LIN {X 0,Y 411.201,Z 389.266,A -85,B 0,C 180,E1 -10586.873,E2 -10586.873} C_VEL
LIN {X 0,Y 411.226,Z 389.263,A -85,B 0,C 180,E1 -10590.644,E2 -10590.644} C_VEL
LIN {X 0,Y 411.231,Z 389.26,A -85,B 0,C 180,E1 -10593.619,E2 -10593.619} C_VEL
LIN {X 0,Y 411.195,Z 389.267,A -85,B 0,C 180,E1 -10596.852,E2 -10596.852} C_VEL
LIN {X 0,Y 411.206,Z 389.262,A -85,B 0,C 180,E1 -10600.05,E2 -10600.05} C_VEL
LIN {X 0,Y 411.255,Z 389.259,A -85,B 0,C 180,E1 -10603.131,E2 -10603.131} C_VEL
LIN {X 0,Y 411.296,Z 389.255,A -85,B 0,C 180,E1 -10606.896,E2 -10606.896} C_VEL
LIN {X 0,Y 411.285,Z 389.254,A -85,B 0,C 180,E1 -10610.161,E2 -10610.161} C_VEL
LIN {X 0,Y 411.447,Z 389.234,A -85,B 0,C 180,E1 -10613.133,E2 -10613.133} C_VEL
LIN {X 0,Y 411.303,Z 389.252,A -85,B 0,C 180,E1 -10615.099,E2 -10615.099} C_VEL
LIN {X 0,Y 411.505,Z 389.226,A -85,B 0,C 180,E1 -10618.043,E2 -10618.043} C_VEL
LIN {X 0,Y 411.635,Z 389.21,A -85,B 0,C 180,E1 -10620,E2 -10620} C_VEL
LIN {X 0,Y 411.458,Z 389.233,A -85,B 0,C 180,E1 -10622.937,E2 -10622.937} C_VEL
LIN {X 0,Y 411.452,Z 389.235,A -85,B 0,C 180,E1 -10626.867,E2 -10626.867} C_VEL
LIN {X 0,Y 411.286,Z 389.253,A -85,B 0,C 180,E1 -10629.839,E2 -10629.839} C_VEL
LIN {X 0,Y 411.297,Z 389.252,A -85,B 0,C 180,E1 -10633.104,E2 -10633.104} C_VEL
LIN {X 0,Y 411.249,Z 389.259,A -85,B 0,C 180,E1 -10636.889,E2 -10636.889} C_VEL
LIN {X 0,Y 411.223,Z 389.262,A -85,B 0,C 180,E1 -10639.987,E2 -10639.987} C_VEL
LIN {X 0,Y 411.196,Z 389.264,A -85,B 0,C 180,E1 -10643.148,E2 -10643.148} C_VEL
LIN {X 0,Y 411.231,Z 389.263,A -85,B 0,C 180,E1 -10646.382,E2 -10646.382} C_VEL
LIN {X 0,Y 411.194,Z 389.265,A -85,B 0,C 180,E1 -10649.713,E2 -10649.713} C_VEL
LIN {X 0,Y 411.201,Z 389.263,A -85,B 0,C 180,E1 -10653.157,E2 -10653.157} C_VEL
LIN {X 0,Y 411.191,Z 389.268,A -85,B 0,C 180,E1 -10656.554,E2 -10656.554} C_VEL
LIN {X 0,Y 411.224,Z 389.262,A -85,B 0,C 180,E1 -10659.731,E2 -10659.731} C_VEL
LIN {X 0,Y 411.173,Z 389.266,A -85,B 0,C 180,E1 -10663.134,E2 -10663.134} C_VEL
LIN {X 0,Y 411.165,Z 389.27,A -85,B 0,C 180,E1 -10665.882,E2 -10665.882} C_VEL
LIN {X 0,Y 411.162,Z 389.269,A -85,B 0,C 180,E1 -10668.772,E2 -10668.772} C_VEL
LIN {X 0,Y 411.209,Z 389.265,A -85,B 0,C 180,E1 -10671.831,E2 -10671.831} C_VEL
LIN {X 0,Y 411.21,Z 389.261,A -85,B 0,C 180,E1 -10675.122,E2 -10675.122} C_VEL
LIN {X 0,Y 411.165,Z 389.272,A -85,B 0,C 180,E1 -10678.004,E2 -10678.004} C_VEL
LIN {X 0,Y 411.218,Z 389.262,A -85,B 0,C 180,E1 -10681.411,E2 -10681.411} C_VEL
LIN {X 0,Y 411.239,Z 389.26,A -85,B 0,C 180,E1 -10683.62,E2 -10683.62} C_VEL
LIN {X 0,Y 411.205,Z 389.262,A -85,B 0,C 180,E1 -10686.853,E2 -10686.853} C_VEL
LIN {X 0,Y 411.217,Z 389.265,A -85,B 0,C 180,E1 -10690.051,E2 -10690.051} C_VEL
LIN {X 0,Y 411.265,Z 389.255,A -85,B 0,C 180,E1 -10693.132,E2 -10693.132} C_VEL
LIN {X 0,Y 411.308,Z 389.249,A -85,B 0,C 180,E1 -10696.896,E2 -10696.896} C_VEL
LIN {X 0,Y 411.295,Z 389.253,A -85,B 0,C 180,E1 -10700.162,E2 -10700.162} C_VEL
LIN {X 0,Y 411.465,Z 389.23,A -85,B 0,C 180,E1 -10703.133,E2 -10703.133} C_VEL
LIN {X 0,Y 411.311,Z 389.25,A -85,B 0,C 180,E1 -10705.099,E2 -10705.099} C_VEL
LIN {X 0,Y 411.438,Z 389.238,A -85,B 0,C 180,E1 -10708.043,E2 -10708.043} C_VEL
LIN {X 0,Y 411.179,Z 389.27,A -85,B 0,C 180,E1 -10710,E2 -10710} C_VEL
LIN {X 0,Y 410.704,Z 389.33,A -85,B 0,C 180,E1 -10710.981,E2 -10710.981} C_VEL
LIN {X 0,Y 410.736,Z 392.015,A -85,B 0,C 180,E1 -10713.925,E2 -10713.925} C_VEL
LIN {X 0,Y 410.647,Z 395.045,A -85,B 0,C 180,E1 -10716.953,E2 -10716.953} C_VEL
LIN {X 0,Y 410.457,Z 397.926,A -85,B 0,C 180,E1 -10719.859,E2 -10719.859} C_VEL
LIN {X 0,Y 410.386,Z 401.01,A -85,B 0,C 180,E1 -10722.864,E2 -10722.864} C_VEL
LIN {X 0,Y 410.342,Z 402.843,A -85,B 0,C 180,E1 -10724.601,E2 -10724.601} C_VEL
LIN {X 0,Y 413.667,Z 416.138,A -85,B 0,C 180,E1 -10725.205,E2 -10725.205} C_VEL
LIN {X 0,Y 415.457,Z 424.901,A -85,B 0,C 180,E1 -10725.704,E2 -10725.704} C_VEL
LIN {X 0,Y 415.437,Z 425.566,A -85,B 0,C 180,E1 -10725.74,E2 -10725.74} C_VEL
LIN {X 0,Y 414.599,Z 431.128,A -85,B 0,C 180,E1 -10726.033,E2 -10726.033} C_VEL
LIN {X 0,Y 411.37,Z 439.883,A -85,B 0,C 180,E1 -10726.51,E2 -10726.51} C_VEL
LIN {X 0,Y 408.025,Z 448.217,A -85,B 0,C 180,E1 -10727.08,E2 -10727.08} C_VEL
LIN {X 0,Y 406.998,Z 453.065,A -85,B 0,C 180,E1 -10727.509,E2 -10727.509} C_VEL
LIN {X 0,Y 406.214,Z 463.524,A -85,B 0,C 180,E1 -10728.667,E2 -10728.667} C_VEL
LIN {X 0,Y 405.456,Z 473.281,A -85,B 0,C 180,E1 -10730.019,E2 -10730.019} C_VEL
LIN {X 0,Y 404.761,Z 481.303,A -85,B 0,C 180,E1 -10731.385,E2 -10731.385} C_VEL
LIN {X 0,Y 404.171,Z 488.245,A -85,B 0,C 180,E1 -10732.838,E2 -10732.838} C_VEL
LIN {X 0,Y 403.811,Z 493.278,A -85,B 0,C 180,E1 -10734.142,E2 -10734.142} C_VEL
LIN {X 0,Y 403.461,Z 498.427,A -85,B 0,C 180,E1 -10735.816,E2 -10735.816} C_VEL
LIN {X 0,Y 403.282,Z 501.804,A -85,B 0,C 180,E1 -10737.279,E2 -10737.279} C_VEL
LIN {X 0,Y 403.135,Z 503.254,A -85,B 0,C 180,E1 -10738.079,E2 -10738.079} C_VEL
LIN {X 0,Y 402.957,Z 504.918,A -85,B 0,C 180,E1 -10739.301,E2 -10739.301} C_VEL
LIN {X 0,Y 402.872,Z 506.388,A -85,B 0,C 180,E1 -10741.263,E2 -10741.263} C_VEL
LIN {X 0,Y 402.872,Z 506.326,A -85,B 0,C 180,E1 -10743.138,E2 -10743.138} C_VEL
LIN {X 0,Y 403.019,Z 504.763,A -85,B 0,C 180,E1 -10745.132,E2 -10745.132} C_VEL
LIN {X 0,Y 403.253,Z 502.375,A -85,B 0,C 180,E1 -10746.707,E2 -10746.707} C_VEL
LIN {X 0,Y 403.549,Z 498.622,A -85,B 0,C 180,E1 -10748.399,E2 -10748.399} C_VEL
LIN {X 0,Y 403.946,Z 493.53,A -85,B 0,C 180,E1 -10750.071,E2 -10750.071} C_VEL
LIN {X 0,Y 404.465,Z 487.306,A -85,B 0,C 180,E1 -10751.654,E2 -10751.654} C_VEL
LIN {X 0,Y 405.136,Z 479.493,A -85,B 0,C 180,E1 -10753.232,E2 -10753.232} C_VEL
LIN {X 0,Y 405.807,Z 471.524,A -85,B 0,C 180,E1 -10754.526,E2 -10754.526} C_VEL
LIN {X 0,Y 406.609,Z 461.592,A -85,B 0,C 180,E1 -10755.831,E2 -10755.831} C_VEL
LIN {X 0,Y 407.402,Z 450.84,A -85,B 0,C 180,E1 -10756.97,E2 -10756.97} C_VEL
LIN {X 0,Y 408.167,Z 439.572,A -85,B 0,C 180,E1 -10757.91,E2 -10757.91} C_VEL
LIN {X 0,Y 408.846,Z 427.215,A -85,B 0,C 180,E1 -10758.702,E2 -10758.702} C_VEL
LIN {X 0,Y 408.184,Z 422.977,A -85,B 0,C 180,E1 -10758.964,E2 -10758.964} C_VEL
LIN {X 0,Y 404.917,Z 410.066,A -85,B 0,C 180,E1 -10759.678,E2 -10759.678} C_VEL
LIN {X 0,Y 403.332,Z 404.392,A -85,B 0,C 180,E1 -10759.963,E2 -10759.963} C_VEL
LIN {X 0,Y 403.388,Z 400.813,A -85,B 0,C 180,E1 -10763.675,E2 -10763.675} C_VEL
LIN {X 0,Y 403.574,Z 397.329,A -85,B 0,C 180,E1 -10767.327,E2 -10767.327} C_VEL
LIN {X 0,Y 403.731,Z 394.082,A -85,B 0,C 180,E1 -10770.829,E2 -10770.829} C_VEL
LIN {X 0,Y 403.781,Z 390.974,A -85,B 0,C 180,E1 -10774.206,E2 -10774.206} C_VEL
LIN {X 0,Y 403.855,Z 390.182,A -85,B 0,C 180,E1 -10775.313,E2 -10775.313} C_VEL
LIN {X 0,Y 404.117,Z 390.153,A -85,B 0,C 180,E1 -10777.505,E2 -10777.505} C_VEL
LIN {X 0,Y 404.161,Z 390.144,A -85,B 0,C 180,E1 -10780.707,E2 -10780.707} C_VEL
LIN {X 0,Y 404.216,Z 390.135,A -85,B 0,C 180,E1 -10783.848,E2 -10783.848} C_VEL
LIN {X 0,Y 404.278,Z 390.129,A -85,B 0,C 180,E1 -10786.939,E2 -10786.939} C_VEL
LIN {X 0,Y 404.254,Z 390.13,A -85,B 0,C 180,E1 -10789.988,E2 -10789.988} C_VEL
LIN {X 0,Y 404.398,Z 390.112,A -85,B 0,C 180,E1 -10793.012,E2 -10793.012} C_VEL
LIN {X 0,Y 404.278,Z 390.125,A -85,B 0,C 180,E1 -10795.013,E2 -10795.013} C_VEL
LIN {X 0,Y 404.477,Z 390.104,A -85,B 0,C 180,E1 -10798.008,E2 -10798.008} C_VEL
LIN {X 0,Y 404.605,Z 390.084,A -85,B 0,C 180,E1 -10800,E2 -10800} C_VEL
LIN {X 0,Y 404.417,Z 390.11,A -85,B 0,C 180,E1 -10802.988,E2 -10802.988} C_VEL
LIN {X 0,Y 404.397,Z 390.112,A -85,B 0,C 180,E1 -10806.987,E2 -10806.987} C_VEL
LIN {X 0,Y 404.253,Z 390.13,A -85,B 0,C 180,E1 -10810.012,E2 -10810.012} C_VEL
LIN {X 0,Y 404.261,Z 390.128,A -85,B 0,C 180,E1 -10813.211,E2 -10813.211} C_VEL
LIN {X 0,Y 404.211,Z 390.135,A -85,B 0,C 180,E1 -10817.007,E2 -10817.007} C_VEL
LIN {X 0,Y 404.159,Z 390.142,A -85,B 0,C 180,E1 -10820.352,E2 -10820.352} C_VEL
LIN {X 0,Y 404.165,Z 390.143,A -85,B 0,C 180,E1 -10823.575,E2 -10823.575} C_VEL
LIN {X 0,Y 404.179,Z 390.14,A -85,B 0,C 180,E1 -10825.767,E2 -10825.767} C_VEL
LIN {X 0,Y 404.191,Z 390.14,A -85,B 0,C 180,E1 -10828,E2 -10828} C_VEL
LIN {X 0,Y 404.135,Z 390.146,A -85,B 0,C 180,E1 -10831.558,E2 -10831.558} C_VEL
LIN {X 0,Y 404.18,Z 390.142,A -85,B 0,C 180,E1 -10835.017,E2 -10835.017} C_VEL
LIN {X 0,Y 404.161,Z 390.144,A -85,B 0,C 180,E1 -10838.756,E2 -10838.756} C_VEL
LIN {X 0,Y 404.147,Z 390.144,A -85,B 0,C 180,E1 -10841.604,E2 -10841.604} C_VEL
LIN {X 0,Y 404.143,Z 390.145,A -85,B 0,C 180,E1 -10844.523,E2 -10844.523} C_VEL
LIN {X 0,Y 404.158,Z 390.285,A -85,B 0,C 180,E1 -10845.838,E2 -10845.838} C_VEL
LIN {X 0,Y 405.078,Z 395.076,A -85,B 0,C 180,E1 -10848.755,E2 -10848.755} C_VEL
LIN {X 0,Y 406.148,Z 401.144,A -85,B 0,C 180,E1 -10852.101,E2 -10852.101} C_VEL
LIN {X 0,Y 406.513,Z 404.837,A -85,B 0,C 180,E1 -10853.999,E2 -10853.999} C_VEL
LIN {X 0,Y 405.924,Z 411.076,A -85,B 0,C 180,E1 -10856.95,E2 -10856.95} C_VEL
LIN {X 0,Y 405.292,Z 418.116,A -85,B 0,C 180,E1 -10860.115,E2 -10860.115} C_VEL
LIN {X 0,Y 404.69,Z 426.478,A -85,B 0,C 180,E1 -10863.715,E2 -10863.715} C_VEL
LIN {X 0,Y 404.135,Z 435.633,A -85,B 0,C 180,E1 -10867.506,E2 -10867.506} C_VEL
LIN {X 0,Y 403.824,Z 443.566,A -85,B 0,C 180,E1 -10870.691,E2 -10870.691} C_VEL
LIN {X 0,Y 403.621,Z 447.012,A -85,B 0,C 180,E1 -10872.063,E2 -10872.063} C_VEL
LIN {X 0,Y 405.834,Z 460.859,A -85,B 0,C 180,E1 -10872.593,E2 -10872.593} C_VEL
LIN {X 0,Y 407.534,Z 473.33,A -85,B 0,C 180,E1 -10873.255,E2 -10873.255} C_VEL
LIN {X 0,Y 407.967,Z 477.581,A -85,B 0,C 180,E1 -10873.516,E2 -10873.516} C_VEL
LIN {X 0,Y 407.145,Z 489.848,A -85,B 0,C 180,E1 -10874.353,E2 -10874.353} C_VEL
LIN {X 0,Y 406.286,Z 501.59,A -85,B 0,C 180,E1 -10875.384,E2 -10875.384} C_VEL
LIN {X 0,Y 405.59,Z 511.467,A -85,B 0,C 180,E1 -10876.472,E2 -10876.472} C_VEL
LIN {X 0,Y 404.871,Z 520.715,A -85,B 0,C 180,E1 -10877.723,E2 -10877.723} C_VEL
LIN {X 0,Y 404.099,Z 529.735,A -85,B 0,C 180,E1 -10879.224,E2 -10879.224} C_VEL
LIN {X 0,Y 403.609,Z 537.015,A -85,B 0,C 180,E1 -10880.731,E2 -10880.731} C_VEL
LIN {X 0,Y 403.301,Z 541.934,A -85,B 0,C 180,E1 -10881.986,E2 -10881.986} C_VEL
LIN {X 0,Y 403.066,Z 547.192,A -85,B 0,C 180,E1 -10883.655,E2 -10883.655} C_VEL
LIN {X 0,Y 403.008,Z 550.396,A -85,B 0,C 180,E1 -10884.998,E2 -10884.998} C_VEL
LIN {X 0,Y 402.878,Z 552.286,A -85,B 0,C 180,E1 -10885.999,E2 -10885.999} C_VEL
LIN {X 0,Y 402.909,Z 553.714,A -85,B 0,C 180,E1 -10887,E2 -10887} C_VEL
LIN {X 0,Y 402.921,Z 554.734,A -85,B 0,C 180,E1 -10888.001,E2 -10888.001} C_VEL
LIN {X 0,Y 402.884,Z 555.359,A -85,B 0,C 180,E1 -10889,E2 -10889} C_VEL
LIN {X 0,Y 402.89,Z 555.588,A -85,B 0,C 180,E1 -10890,E2 -10890} C_VEL
LIN {X 0,Y 402.884,Z 555.376,A -85,B 0,C 180,E1 -10890.999,E2 -10890.999} C_VEL
LIN {X 0,Y 402.921,Z 554.772,A -85,B 0,C 180,E1 -10891.999,E2 -10891.999} C_VEL
LIN {X 0,Y 402.909,Z 553.771,A -85,B 0,C 180,E1 -10892.999,E2 -10892.999} C_VEL
LIN {X 0,Y 402.877,Z 552.361,A -85,B 0,C 180,E1 -10894.001,E2 -10894.001} C_VEL
LIN {X 0,Y 403.006,Z 549.406,A -85,B 0,C 180,E1 -10895.504,E2 -10895.504} C_VEL
LIN {X 0,Y 403.116,Z 545.396,A -85,B 0,C 180,E1 -10897.009,E2 -10897.009} C_VEL
LIN {X 0,Y 403.516,Z 539.236,A -85,B 0,C 180,E1 -10898.765,E2 -10898.765} C_VEL
LIN {X 0,Y 403.964,Z 532.509,A -85,B 0,C 180,E1 -10900.272,E2 -10900.272} C_VEL
LIN {X 0,Y 404.586,Z 524.172,A -85,B 0,C 180,E1 -10901.777,E2 -10901.777} C_VEL
LIN {X 0,Y 405.266,Z 515.622,A -85,B 0,C 180,E1 -10903.028,E2 -10903.028} C_VEL
LIN {X 0,Y 406.019,Z 505.572,A -85,B 0,C 180,E1 -10904.225,E2 -10904.225} C_VEL
LIN {X 0,Y 406.801,Z 494.649,A -85,B 0,C 180,E1 -10905.275,E2 -10905.275} C_VEL
LIN {X 0,Y 407.651,Z 483.346,A -85,B 0,C 180,E1 -10906.133,E2 -10906.133} C_VEL
LIN {X 0,Y 407.972,Z 476.714,A -85,B 0,C 180,E1 -10906.544,E2 -10906.544} C_VEL
LIN {X 0,Y 406.146,Z 463.38,A -85,B 0,C 180,E1 -10907.286,E2 -10907.286} C_VEL
LIN {X 0,Y 404.097,Z 450.537,A -85,B 0,C 180,E1 -10907.811,E2 -10907.811} C_VEL
LIN {X 0,Y 403.641,Z 447.507,A -85,B 0,C 180,E1 -10907.936,E2 -10907.936} C_VEL
LIN {X 0,Y 404.08,Z 438.83,A -85,B 0,C 180,E1 -10911.422,E2 -10911.422} C_VEL
LIN {X 0,Y 404.484,Z 430.976,A -85,B 0,C 180,E1 -10914.645,E2 -10914.645} C_VEL
LIN {X 0,Y 405.044,Z 423.172,A -85,B 0,C 180,E1 -10917.935,E2 -10917.935} C_VEL
LIN {X 0,Y 405.766,Z 414.008,A -85,B 0,C 180,E1 -10921.93,E2 -10921.93} C_VEL
LIN {X 0,Y 406.342,Z 407.661,A -85,B 0,C 180,E1 -10924.802,E2 -10924.802} C_VEL
LIN {X 0,Y 406.521,Z 403.834,A -85,B 0,C 180,E1 -10926.614,E2 -10926.614} C_VEL
LIN {X 0,Y 405.706,Z 398.526,A -85,B 0,C 180,E1 -10929.291,E2 -10929.291} C_VEL
LIN {X 0,Y 404.537,Z 392.321,A -85,B 0,C 180,E1 -10932.651,E2 -10932.651} C_VEL
LIN {X 0,Y 404.127,Z 390.147,A -85,B 0,C 180,E1 -10933.89,E2 -10933.89} C_VEL
LIN {X 0,Y 404.166,Z 390.143,A -85,B 0,C 180,E1 -10937.299,E2 -10937.299} C_VEL
LIN {X 0,Y 404.163,Z 390.142,A -85,B 0,C 180,E1 -10939.955,E2 -10939.955} C_VEL
LIN {X 0,Y 404.135,Z 390.146,A -85,B 0,C 180,E1 -10943.123,E2 -10943.123} C_VEL
LIN {X 0,Y 404.138,Z 390.143,A -85,B 0,C 180,E1 -10946.187,E2 -10946.187} C_VEL
LIN {X 0,Y 404.138,Z 390.142,A -85,B 0,C 180,E1 -10949.714,E2 -10949.714} C_VEL
LIN {X 0,Y 404.188,Z 390.139,A -85,B 0,C 180,E1 -10953.122,E2 -10953.122} C_VEL
LIN {X 0,Y 404.169,Z 390.14,A -85,B 0,C 180,E1 -10955.334,E2 -10955.334} C_VEL
LIN {X 0,Y 404.131,Z 390.147,A -85,B 0,C 180,E1 -10958.58,E2 -10958.58} C_VEL
LIN {X 0,Y 404.202,Z 390.134,A -85,B 0,C 180,E1 -10961.762,E2 -10961.762} C_VEL
LIN {X 0,Y 404.197,Z 390.139,A -85,B 0,C 180,E1 -10964.882,E2 -10964.882} C_VEL
LIN {X 0,Y 404.248,Z 390.128,A -85,B 0,C 180,E1 -10967.958,E2 -10967.958} C_VEL
LIN {X 0,Y 404.396,Z 390.112,A -85,B 0,C 180,E1 -10972.129,E2 -10972.129} C_VEL
LIN {X 0,Y 404.414,Z 390.109,A -85,B 0,C 180,E1 -10974.015,E2 -10974.015} C_VEL
LIN {X 0,Y 404.474,Z 390.101,A -85,B 0,C 180,E1 -10978.009,E2 -10978.009} C_VEL
LIN {X 0,Y 404.604,Z 390.085,A -85,B 0,C 180,E1 -10980,E2 -10980} C_VEL
LIN {X 0,Y 404.415,Z 390.11,A -85,B 0,C 180,E1 -10982.989,E2 -10982.989} C_VEL
LIN {X 0,Y 404.403,Z 390.111,A -85,B 0,C 180,E1 -10986.988,E2 -10986.988} C_VEL
LIN {X 0,Y 404.251,Z 390.13,A -85,B 0,C 180,E1 -10990.012,E2 -10990.012} C_VEL
LIN {X 0,Y 404.258,Z 390.128,A -85,B 0,C 180,E1 -10993.212,E2 -10993.212} C_VEL
LIN {X 0,Y 404.208,Z 390.135,A -85,B 0,C 180,E1 -10997.008,E2 -10997.008} C_VEL
LIN {X 0,Y 404.156,Z 390.144,A -85,B 0,C 180,E1 -11000.352,E2 -11000.352} C_VEL
LIN {X 0,Y 404.162,Z 390.139,A -85,B 0,C 180,E1 -11003.575,E2 -11003.575} C_VEL
LIN {X 0,Y 404.177,Z 390.138,A -85,B 0,C 180,E1 -11005.767,E2 -11005.767} C_VEL
LIN {X 0,Y 404.189,Z 390.139,A -85,B 0,C 180,E1 -11008,E2 -11008} C_VEL
LIN {X 0,Y 404.133,Z 390.143,A -85,B 0,C 180,E1 -11011.559,E2 -11011.559} C_VEL
LIN {X 0,Y 404.18,Z 390.137,A -85,B 0,C 180,E1 -11015.017,E2 -11015.017} C_VEL
LIN {X 0,Y 404.159,Z 390.141,A -85,B 0,C 180,E1 -11018.757,E2 -11018.757} C_VEL
LIN {X 0,Y 404.146,Z 390.143,A -85,B 0,C 180,E1 -11021.605,E2 -11021.605} C_VEL
LIN {X 0,Y 404.141,Z 390.145,A -85,B 0,C 180,E1 -11024.523,E2 -11024.523} C_VEL
LIN {X 0,Y 404.133,Z 390.143,A -85,B 0,C 180,E1 -11027.297,E2 -11027.297} C_VEL
LIN {X 0,Y 404.166,Z 390.142,A -85,B 0,C 180,E1 -11029.956,E2 -11029.956} C_VEL
LIN {X 0,Y 404.138,Z 390.142,A -85,B 0,C 180,E1 -11033.125,E2 -11033.125} C_VEL
LIN {X 0,Y 404.144,Z 390.145,A -85,B 0,C 180,E1 -11036.189,E2 -11036.189} C_VEL
LIN {X 0,Y 404.145,Z 390.145,A -85,B 0,C 180,E1 -11039.716,E2 -11039.716} C_VEL
LIN {X 0,Y 404.196,Z 390.135,A -85,B 0,C 180,E1 -11043.124,E2 -11043.124} C_VEL
LIN {X 0,Y 404.178,Z 390.138,A -85,B 0,C 180,E1 -11045.335,E2 -11045.335} C_VEL
LIN {X 0,Y 404.141,Z 390.143,A -85,B 0,C 180,E1 -11048.581,E2 -11048.581} C_VEL
LIN {X 0,Y 404.212,Z 390.137,A -85,B 0,C 180,E1 -11051.763,E2 -11051.763} C_VEL
LIN {X 0,Y 404.209,Z 390.133,A -85,B 0,C 180,E1 -11054.883,E2 -11054.883} C_VEL
LIN {X 0,Y 404.259,Z 390.131,A -85,B 0,C 180,E1 -11057.959,E2 -11057.959} C_VEL
LIN {X 0,Y 404.437,Z 390.108,A -85,B 0,C 180,E1 -11062.1,E2 -11062.1} C_VEL
LIN {X 0,Y 404.428,Z 390.11,A -85,B 0,C 180,E1 -11064.016,E2 -11064.016} C_VEL
LIN {X 0,Y 404.405,Z 390.114,A -85,B 0,C 180,E1 -11068.008,E2 -11068.008} C_VEL
LIN {X 0,Y 404.14,Z 390.146,A -85,B 0,C 180,E1 -11070,E2 -11070} C_VEL
LIN {X 0,Y 403.648,Z 390.209,A -85,B 0,C 180,E1 -11070.998,E2 -11070.998} C_VEL
LIN {X 0,Y 403.695,Z 392.899,A -85,B 0,C 180,E1 -11073.993,E2 -11073.993} C_VEL
LIN {X 0,Y 403.592,Z 395.857,A -85,B 0,C 180,E1 -11077.002,E2 -11077.002} C_VEL
LIN {X 0,Y 403.408,Z 398.919,A -85,B 0,C 180,E1 -11080.033,E2 -11080.033} C_VEL
LIN {X 0,Y 403.316,Z 401.99,A -85,B 0,C 180,E1 -11083.093,E2 -11083.093} C_VEL
LIN {X 0,Y 403.283,Z 403.217,A -85,B 0,C 180,E1 -11084.282,E2 -11084.282} C_VEL
LIN {X 0,Y 407.061,Z 418.238,A -85,B 0,C 180,E1 -11085.009,E2 -11085.009} C_VEL
LIN {X 0,Y 408.554,Z 426.223,A -85,B 0,C 180,E1 -11085.485,E2 -11085.485} C_VEL
LIN {X 0,Y 407.925,Z 438.431,A -85,B 0,C 180,E1 -11086.258,E2 -11086.258} C_VEL
LIN {X 0,Y 407.244,Z 449.754,A -85,B 0,C 180,E1 -11087.189,E2 -11087.189} C_VEL
LIN {X 0,Y 406.998,Z 453.065,A -85,B 0,C 180,E1 -11087.509,E2 -11087.509} C_VEL
LIN {X 0,Y 406.095,Z 456.322,A -85,B 0,C 180,E1 -11087.81,E2 -11087.81} C_VEL
LIN {X 0,Y 402.946,Z 461.386,A -85,B 0,C 180,E1 -11088.262,E2 -11088.262} C_VEL
LIN {X 0,Y 399.796,Z 466.214,A -85,B 0,C 180,E1 -11088.763,E2 -11088.763} C_VEL
LIN {X 0,Y 398.895,Z 469.097,A -85,B 0,C 180,E1 -11089.135,E2 -11089.135} C_VEL
LIN {X 0,Y 398.052,Z 478.873,A -85,B 0,C 180,E1 -11090.678,E2 -11090.678} C_VEL
LIN {X 0,Y 397.414,Z 485.971,A -85,B 0,C 180,E1 -11092.073,E2 -11092.073} C_VEL
LIN {X 0,Y 396.868,Z 492.79,A -85,B 0,C 180,E1 -11093.757,E2 -11093.757} C_VEL
LIN {X 0,Y 396.454,Z 497.701,A -85,B 0,C 180,E1 -11095.299,E2 -11095.299} C_VEL
LIN {X 0,Y 396.27,Z 501.565,A -85,B 0,C 180,E1 -11096.888,E2 -11096.888} C_VEL
LIN {X 0,Y 395.955,Z 504.581,A -85,B 0,C 180,E1 -11098.635,E2 -11098.635} C_VEL
LIN {X 0,Y 395.838,Z 505.909,A -85,B 0,C 180,E1 -11099.81,E2 -11099.81} C_VEL
LIN {X 0,Y 395.792,Z 506.878,A -85,B 0,C 180,E1 -11101.534,E2 -11101.534} C_VEL
LIN {X 0,Y 395.804,Z 506.646,A -85,B 0,C 180,E1 -11103.431,E2 -11103.431} C_VEL
LIN {X 0,Y 395.951,Z 505.129,A -85,B 0,C 180,E1 -11105.265,E2 -11105.265} C_VEL
LIN {X 0,Y 396.224,Z 502.271,A -85,B 0,C 180,E1 -11107.09,E2 -11107.09} C_VEL
LIN {X 0,Y 396.547,Z 498.426,A -85,B 0,C 180,E1 -11108.756,E2 -11108.756} C_VEL
LIN {X 0,Y 397,Z 493.255,A -85,B 0,C 180,E1 -11110.428,E2 -11110.428} C_VEL
LIN {X 0,Y 397.567,Z 486.778,A -85,B 0,C 180,E1 -11112.058,E2 -11112.058} C_VEL
LIN {X 0,Y 398.22,Z 479.634,A -85,B 0,C 180,E1 -11113.494,E2 -11113.494} C_VEL
LIN {X 0,Y 398.951,Z 471.653,A -85,B 0,C 180,E1 -11114.8,E2 -11114.8} C_VEL
LIN {X 0,Y 399.782,Z 461.765,A -85,B 0,C 180,E1 -11116.117,E2 -11116.117} C_VEL
LIN {X 0,Y 400.59,Z 451.383,A -85,B 0,C 180,E1 -11117.232,E2 -11117.232} C_VEL
LIN {X 0,Y 401.38,Z 440.025,A -85,B 0,C 180,E1 -11118.197,E2 -11118.197} C_VEL
LIN {X 0,Y 402.026,Z 427.13,A -85,B 0,C 180,E1 -11119.037,E2 -11119.037} C_VEL
LIN {X 0,Y 399.081,Z 414.809,A -85,B 0,C 180,E1 -11119.792,E2 -11119.792} C_VEL
LIN {X 0,Y 396.252,Z 404.877,A -85,B 0,C 180,E1 -11120.282,E2 -11120.282} C_VEL
LIN {X 0,Y 396.31,Z 402.335,A -85,B 0,C 180,E1 -11122.939,E2 -11122.939} C_VEL
LIN {X 0,Y 396.521,Z 398.814,A -85,B 0,C 180,E1 -11126.67,E2 -11126.67} C_VEL
LIN {X 0,Y 396.627,Z 395.514,A -85,B 0,C 180,E1 -11130.255,E2 -11130.255} C_VEL
LIN {X 0,Y 396.718,Z 392.384,A -85,B 0,C 180,E1 -11133.712,E2 -11133.712} C_VEL
LIN {X 0,Y 396.79,Z 391.365,A -85,B 0,C 180,E1 -11134.843,E2 -11134.843} C_VEL
LIN {X 0,Y 397.01,Z 391.039,A -85,B 0,C 180,E1 -11137.079,E2 -11137.079} C_VEL
LIN {X 0,Y 397.143,Z 391.018,A -85,B 0,C 180,E1 -11140.352,E2 -11140.352} C_VEL
LIN {X 0,Y 397.162,Z 391.015,A -85,B 0,C 180,E1 -11143.553,E2 -11143.553} C_VEL
LIN {X 0,Y 397.224,Z 391.008,A -85,B 0,C 180,E1 -11146.702,E2 -11146.702} C_VEL
LIN {X 0,Y 397.213,Z 391.008,A -85,B 0,C 180,E1 -11149.809,E2 -11149.809} C_VEL
LIN {X 0,Y 397.347,Z 390.99,A -85,B 0,C 180,E1 -11152.888,E2 -11152.888} C_VEL
LIN {X 0,Y 397.25,Z 391,A -85,B 0,C 180,E1 -11154.925,E2 -11154.925} C_VEL
LIN {X 0,Y 397.446,Z 390.979,A -85,B 0,C 180,E1 -11157.973,E2 -11157.973} C_VEL
LIN {X 0,Y 397.575,Z 390.96,A -85,B 0,C 180,E1 -11160,E2 -11160} C_VEL
LIN {X 0,Y 397.376,Z 390.988,A -85,B 0,C 180,E1 -11163.041,E2 -11163.041} C_VEL
LIN {X 0,Y 397.368,Z 390.988,A -85,B 0,C 180,E1 -11166.092,E2 -11166.092} C_VEL
LIN {X 0,Y 397.248,Z 391.004,A -85,B 0,C 180,E1 -11169.162,E2 -11169.162} C_VEL
LIN {X 0,Y 397.214,Z 391.008,A -85,B 0,C 180,E1 -11172.258,E2 -11172.258} C_VEL
LIN {X 0,Y 397.173,Z 391.011,A -85,B 0,C 180,E1 -11175.392,E2 -11175.392} C_VEL
LIN {X 0,Y 397.157,Z 391.012,A -85,B 0,C 180,E1 -11178.574,E2 -11178.574} C_VEL
LIN {X 0,Y 397.092,Z 391.023,A -85,B 0,C 180,E1 -11181.819,E2 -11181.819} C_VEL
LIN {X 0,Y 397.152,Z 391.015,A -85,B 0,C 180,E1 -11185.132,E2 -11185.132} C_VEL
LIN {X 0,Y 397.158,Z 391.015,A -85,B 0,C 180,E1 -11187.776,E2 -11187.776} C_VEL
LIN {X 0,Y 397.074,Z 391.025,A -85,B 0,C 180,E1 -11190.883,E2 -11190.883} C_VEL
LIN {X 0,Y 397.121,Z 391.022,A -85,B 0,C 180,E1 -11194.494,E2 -11194.494} C_VEL
LIN {X 0,Y 397.107,Z 391.023,A -85,B 0,C 180,E1 -11198.275,E2 -11198.275} C_VEL
LIN {X 0,Y 397.11,Z 391.022,A -85,B 0,C 180,E1 -11200.906,E2 -11200.906} C_VEL
LIN {X 0,Y 397.1,Z 391.023,A -85,B 0,C 180,E1 -11203.649,E2 -11203.649} C_VEL
LIN {X 0,Y 397.121,Z 391.179,A -85,B 0,C 180,E1 -11205.424,E2 -11205.424} C_VEL
LIN {X 0,Y 398.083,Z 396.207,A -85,B 0,C 180,E1 -11208.576,E2 -11208.576} C_VEL
LIN {X 0,Y 399.273,Z 402.981,A -85,B 0,C 180,E1 -11212.381,E2 -11212.381} C_VEL
LIN {X 0,Y 399.501,Z 406.142,A -85,B 0,C 180,E1 -11214.021,E2 -11214.021} C_VEL
LIN {X 0,Y 398.917,Z 412.113,A -85,B 0,C 180,E1 -11216.897,E2 -11216.897} C_VEL
LIN {X 0,Y 398.328,Z 418.509,A -85,B 0,C 180,E1 -11219.831,E2 -11219.831} C_VEL
LIN {X 0,Y 397.715,Z 426.148,A -85,B 0,C 180,E1 -11223.218,E2 -11223.218} C_VEL
LIN {X 0,Y 397.124,Z 435.266,A -85,B 0,C 180,E1 -11227.087,E2 -11227.087} C_VEL
LIN {X 0,Y 396.725,Z 444.455,A -85,B 0,C 180,E1 -11230.869,E2 -11230.869} C_VEL
LIN {X 0,Y 396.601,Z 446.727,A -85,B 0,C 180,E1 -11231.734,E2 -11231.734} C_VEL
LIN {X 0,Y 398.859,Z 460.567,A -85,B 0,C 180,E1 -11232.275,E2 -11232.275} C_VEL
LIN {X 0,Y 400.467,Z 472.664,A -85,B 0,C 180,E1 -11232.93,E2 -11232.93} C_VEL
LIN {X 0,Y 401.086,Z 477.63,A -85,B 0,C 180,E1 -11233.25,E2 -11233.25} C_VEL
LIN {X 0,Y 400.301,Z 489.47,A -85,B 0,C 180,E1 -11234.078,E2 -11234.078} C_VEL
LIN {X 0,Y 399.381,Z 501.182,A -85,B 0,C 180,E1 -11235.126,E2 -11235.126} C_VEL
LIN {X 0,Y 398.624,Z 511.375,A -85,B 0,C 180,E1 -11236.275,E2 -11236.275} C_VEL
LIN {X 0,Y 397.915,Z 520.275,A -85,B 0,C 180,E1 -11237.505,E2 -11237.505} C_VEL
LIN {X 0,Y 397.087,Z 529.295,A -85,B 0,C 180,E1 -11239.032,E2 -11239.032} C_VEL
LIN {X 0,Y 396.565,Z 536.576,A -85,B 0,C 180,E1 -11240.565,E2 -11240.565} C_VEL
LIN {X 0,Y 396.243,Z 541.498,A -85,B 0,C 180,E1 -11241.843,E2 -11241.843} C_VEL
LIN {X 0,Y 395.993,Z 547.054,A -85,B 0,C 180,E1 -11243.657,E2 -11243.657} C_VEL
LIN {X 0,Y 395.921,Z 549.963,A -85,B 0,C 180,E1 -11244.908,E2 -11244.908} C_VEL
LIN {X 0,Y 395.803,Z 551.855,A -85,B 0,C 180,E1 -11245.927,E2 -11245.927} C_VEL
LIN {X 0,Y 395.813,Z 553.281,A -85,B 0,C 180,E1 -11246.946,E2 -11246.946} C_VEL
LIN {X 0,Y 395.854,Z 554.305,A -85,B 0,C 180,E1 -11247.965,E2 -11247.965} C_VEL
LIN {X 0,Y 395.813,Z 554.931,A -85,B 0,C 180,E1 -11248.982,E2 -11248.982} C_VEL
LIN {X 0,Y 395.815,Z 555.159,A -85,B 0,C 180,E1 -11250,E2 -11250} C_VEL
LIN {X 0,Y 395.813,Z 554.947,A -85,B 0,C 180,E1 -11251.017,E2 -11251.017} C_VEL
LIN {X 0,Y 395.854,Z 554.343,A -85,B 0,C 180,E1 -11252.035,E2 -11252.035} C_VEL
LIN {X 0,Y 395.812,Z 553.341,A -85,B 0,C 180,E1 -11253.053,E2 -11253.053} C_VEL
LIN {X 0,Y 395.802,Z 551.93,A -85,B 0,C 180,E1 -11254.073,E2 -11254.073} C_VEL
LIN {X 0,Y 395.907,Z 548.972,A -85,B 0,C 180,E1 -11255.603,E2 -11255.603} C_VEL
LIN {X 0,Y 396.061,Z 544.961,A -85,B 0,C 180,E1 -11257.135,E2 -11257.135} C_VEL
LIN {X 0,Y 396.457,Z 538.795,A -85,B 0,C 180,E1 -11258.923,E2 -11258.923} C_VEL
LIN {X 0,Y 396.912,Z 532.064,A -85,B 0,C 180,E1 -11260.456,E2 -11260.456} C_VEL
LIN {X 0,Y 397.581,Z 523.724,A -85,B 0,C 180,E1 -11261.987,E2 -11261.987} C_VEL
LIN {X 0,Y 398.304,Z 515.169,A -85,B 0,C 180,E1 -11263.26,E2 -11263.26} C_VEL
LIN {X 0,Y 399.109,Z 504.851,A -85,B 0,C 180,E1 -11264.506,E2 -11264.506} C_VEL
LIN {X 0,Y 399.932,Z 494.187,A -85,B 0,C 180,E1 -11265.544,E2 -11265.544} C_VEL
LIN {X 0,Y 400.808,Z 482.97,A -85,B 0,C 180,E1 -11266.409,E2 -11266.409} C_VEL
LIN {X 0,Y 401.08,Z 477.723,A -85,B 0,C 180,E1 -11266.747,E2 -11266.747} C_VEL
LIN {X 0,Y 399.405,Z 464.941,A -85,B 0,C 180,E1 -11267.496,E2 -11267.496} C_VEL
LIN {X 0,Y 397.258,Z 451.327,A -85,B 0,C 180,E1 -11268.084,E2 -11268.084} C_VEL
LIN {X 0,Y 396.605,Z 447.191,A -85,B 0,C 180,E1 -11268.232,E2 -11268.232} C_VEL
LIN {X 0,Y 397.045,Z 438.464,A -85,B 0,C 180,E1 -11271.821,E2 -11271.821} C_VEL
LIN {X 0,Y 397.624,Z 429.367,A -85,B 0,C 180,E1 -11275.654,E2 -11275.654} C_VEL
LIN {X 0,Y 398.189,Z 421.539,A -85,B 0,C 180,E1 -11279.036,E2 -11279.036} C_VEL
LIN {X 0,Y 398.772,Z 414.453,A -85,B 0,C 180,E1 -11282.225,E2 -11282.225} C_VEL
LIN {X 0,Y 399.467,Z 407.409,A -85,B 0,C 180,E1 -11285.49,E2 -11285.49} C_VEL
LIN {X 0,Y 399.516,Z 404.85,A -85,B 0,C 180,E1 -11286.733,E2 -11286.733} C_VEL
LIN {X 0,Y 398.721,Z 399.706,A -85,B 0,C 180,E1 -11289.385,E2 -11289.385} C_VEL
LIN {X 0,Y 397.523,Z 393.426,A -85,B 0,C 180,E1 -11292.845,E2 -11292.845} C_VEL
LIN {X 0,Y 397.098,Z 391.024,A -85,B 0,C 180,E1 -11294.267,E2 -11294.267} C_VEL
LIN {X 0,Y 397.109,Z 391.021,A -85,B 0,C 180,E1 -11297.738,E2 -11297.738} C_VEL
LIN {X 0,Y 397.132,Z 391.019,A -85,B 0,C 180,E1 -11301.136,E2 -11301.136} C_VEL
LIN {X 0,Y 397.114,Z 391.019,A -85,B 0,C 180,E1 -11304.496,E2 -11304.496} C_VEL
LIN {X 0,Y 397.071,Z 391.022,A -85,B 0,C 180,E1 -11307.928,E2 -11307.928} C_VEL
LIN {X 0,Y 397.115,Z 391.018,A -85,B 0,C 180,E1 -11311.456,E2 -11311.456} C_VEL
LIN {X 0,Y 397.145,Z 391.016,A -85,B 0,C 180,E1 -11314.487,E2 -11314.487} C_VEL
LIN {X 0,Y 397.101,Z 391.022,A -85,B 0,C 180,E1 -11317.085,E2 -11317.085} C_VEL
LIN {X 0,Y 397.14,Z 391.016,A -85,B 0,C 180,E1 -11320.352,E2 -11320.352} C_VEL
LIN {X 0,Y 397.158,Z 391.012,A -85,B 0,C 180,E1 -11323.553,E2 -11323.553} C_VEL
LIN {X 0,Y 397.22,Z 391.008,A -85,B 0,C 180,E1 -11326.702,E2 -11326.702} C_VEL
LIN {X 0,Y 397.21,Z 391.005,A -85,B 0,C 180,E1 -11329.809,E2 -11329.809} C_VEL
LIN {X 0,Y 397.344,Z 390.992,A -85,B 0,C 180,E1 -11332.888,E2 -11332.888} C_VEL
LIN {X 0,Y 397.247,Z 391.004,A -85,B 0,C 180,E1 -11334.925,E2 -11334.925} C_VEL
LIN {X 0,Y 397.443,Z 390.977,A -85,B 0,C 180,E1 -11337.973,E2 -11337.973} C_VEL
LIN {X 0,Y 397.574,Z 390.961,A -85,B 0,C 180,E1 -11340,E2 -11340} C_VEL
LIN {X 0,Y 397.374,Z 390.987,A -85,B 0,C 180,E1 -11343.042,E2 -11343.042} C_VEL
LIN {X 0,Y 397.355,Z 390.988,A -85,B 0,C 180,E1 -11347.112,E2 -11347.112} C_VEL
LIN {X 0,Y 397.211,Z 391.008,A -85,B 0,C 180,E1 -11350.191,E2 -11350.191} C_VEL
LIN {X 0,Y 397.218,Z 391.004,A -85,B 0,C 180,E1 -11353.321,E2 -11353.321} C_VEL
LIN {X 0,Y 397.174,Z 391.01,A -85,B 0,C 180,E1 -11357.156,E2 -11357.156} C_VEL
LIN {X 0,Y 397.095,Z 391.023,A -85,B 0,C 180,E1 -11360.731,E2 -11360.731} C_VEL
LIN {X 0,Y 397.126,Z 391.018,A -85,B 0,C 180,E1 -11364.019,E2 -11364.019} C_VEL
LIN {X 0,Y 397.188,Z 391.008,A -85,B 0,C 180,E1 -11367.391,E2 -11367.391} C_VEL
LIN {X 0,Y 397.072,Z 391.024,A -85,B 0,C 180,E1 -11370.883,E2 -11370.883} C_VEL
LIN {X 0,Y 397.121,Z 391.02,A -85,B 0,C 180,E1 -11374.494,E2 -11374.494} C_VEL
LIN {X 0,Y 397.106,Z 391.023,A -85,B 0,C 180,E1 -11378.275,E2 -11378.275} C_VEL
LIN {X 0,Y 397.109,Z 391.018,A -85,B 0,C 180,E1 -11380.907,E2 -11380.907} C_VEL
LIN {X 0,Y 397.098,Z 391.02,A -85,B 0,C 180,E1 -11383.649,E2 -11383.649} C_VEL
LIN {X 0,Y 397.099,Z 391.022,A -85,B 0,C 180,E1 -11386.522,E2 -11386.522} C_VEL
LIN {X 0,Y 397.113,Z 391.02,A -85,B 0,C 180,E1 -11390.424,E2 -11390.424} C_VEL
LIN {X 0,Y 397.108,Z 391.022,A -85,B 0,C 180,E1 -11394.266,E2 -11394.266} C_VEL
LIN {X 0,Y 397.114,Z 391.018,A -85,B 0,C 180,E1 -11396.728,E2 -11396.728} C_VEL
LIN {X 0,Y 397.124,Z 391.019,A -85,B 0,C 180,E1 -11400.297,E2 -11400.297} C_VEL
LIN {X 0,Y 397.195,Z 391.007,A -85,B 0,C 180,E1 -11402.611,E2 -11402.611} C_VEL
LIN {X 0,Y 397.134,Z 391.019,A -85,B 0,C 180,E1 -11405.983,E2 -11405.983} C_VEL
LIN {X 0,Y 397.14,Z 391.018,A -85,B 0,C 180,E1 -11409.705,E2 -11409.705} C_VEL
LIN {X 0,Y 397.184,Z 391.008,A -85,B 0,C 180,E1 -11412.846,E2 -11412.846} C_VEL
LIN {X 0,Y 397.231,Z 391.003,A -85,B 0,C 180,E1 -11416.703,E2 -11416.703} C_VEL
LIN {X 0,Y 397.22,Z 391.008,A -85,B 0,C 180,E1 -11419.81,E2 -11419.81} C_VEL
LIN {X 0,Y 397.368,Z 390.985,A -85,B 0,C 180,E1 -11422.889,E2 -11422.889} C_VEL
LIN {X 0,Y 397.256,Z 391,A -85,B 0,C 180,E1 -11424.926,E2 -11424.926} C_VEL
LIN {X 0,Y 397.371,Z 390.99,A -85,B 0,C 180,E1 -11427.973,E2 -11427.973} C_VEL
LIN {X 0,Y 397.101,Z 391.023,A -85,B 0,C 180,E1 -11430,E2 -11430} C_VEL
LIN {X 0,Y 396.592,Z 391.088,A -85,B 0,C 180,E1 -11431.016,E2 -11431.016} C_VEL
LIN {X 0,Y 396.654,Z 393.764,A -85,B 0,C 180,E1 -11434.064,E2 -11434.064} C_VEL
LIN {X 0,Y 396.537,Z 396.742,A -85,B 0,C 180,E1 -11437.127,E2 -11437.127} C_VEL
LIN {X 0,Y 396.345,Z 399.838,A -85,B 0,C 180,E1 -11440.214,E2 -11440.214} C_VEL
LIN {X 0,Y 396.243,Z 402.999,A -85,B 0,C 180,E1 -11443.331,E2 -11443.331} C_VEL
LIN {X 0,Y 396.226,Z 403.661,A -85,B 0,C 180,E1 -11443.985,E2 -11443.985} C_VEL
LIN {X 0,Y 399.623,Z 417.032,A -85,B 0,C 180,E1 -11444.624,E2 -11444.624} C_VEL
LIN {X 0,Y 401.756,Z 426.68,A -85,B 0,C 180,E1 -11445.212,E2 -11445.212} C_VEL
LIN {X 0,Y 401.112,Z 438.8,A -85,B 0,C 180,E1 -11445.993,E2 -11445.993} C_VEL
LIN {X 0,Y 400.35,Z 450.439,A -85,B 0,C 180,E1 -11446.968,E2 -11446.968} C_VEL
LIN {X 0,Y 399.466,Z 461.802,A -85,B 0,C 180,E1 -11448.185,E2 -11448.185} C_VEL
LIN {X 0,Y 398.895,Z 469.097,A -85,B 0,C 180,E1 -11449.135,E2 -11449.135} C_VEL
LIN {X 0,Y 397.879,Z 473.278,A -85,B 0,C 180,E1 -11449.725,E2 -11449.725} C_VEL
LIN {X 0,Y 394.481,Z 479.723,A -85,B 0,C 180,E1 -11450.696,E2 -11450.696} C_VEL
LIN {X 0,Y 391.128,Z 485.606,A -85,B 0,C 180,E1 -11451.753,E2 -11451.753} C_VEL
LIN {X 0,Y 390.196,Z 488.815,A -85,B 0,C 180,E1 -11452.467,E2 -11452.467} C_VEL
LIN {X 0,Y 389.761,Z 494.317,A -85,B 0,C 180,E1 -11453.935,E2 -11453.935} C_VEL
LIN {X 0,Y 389.34,Z 499.422,A -85,B 0,C 180,E1 -11455.672,E2 -11455.672} C_VEL
LIN {X 0,Y 389.196,Z 502.056,A -85,B 0,C 180,E1 -11456.836,E2 -11456.836} C_VEL
LIN {X 0,Y 388.963,Z 504.208,A -85,B 0,C 180,E1 -11458.02,E2 -11458.02} C_VEL
LIN {X 0,Y 388.753,Z 506.356,A -85,B 0,C 180,E1 -11459.8,E2 -11459.8} C_VEL
LIN {X 0,Y 388.707,Z 507.363,A -85,B 0,C 180,E1 -11461.811,E2 -11461.811} C_VEL
LIN {X 0,Y 388.745,Z 506.965,A -85,B 0,C 180,E1 -11463.734,E2 -11463.734} C_VEL
LIN {X 0,Y 388.925,Z 505.24,A -85,B 0,C 180,E1 -11465.593,E2 -11465.593} C_VEL
LIN {X 0,Y 389.217,Z 502.312,A -85,B 0,C 180,E1 -11467.392,E2 -11467.392} C_VEL
LIN {X 0,Y 389.594,Z 498.163,A -85,B 0,C 180,E1 -11469.151,E2 -11469.151} C_VEL
LIN {X 0,Y 390.067,Z 492.909,A -85,B 0,C 180,E1 -11470.823,E2 -11470.823} C_VEL
LIN {X 0,Y 390.685,Z 486.211,A -85,B 0,C 180,E1 -11472.477,E2 -11472.477} C_VEL
LIN {X 0,Y 391.492,Z 477.87,A -85,B 0,C 180,E1 -11474.104,E2 -11474.104} C_VEL
LIN {X 0,Y 392.282,Z 469.726,A -85,B 0,C 180,E1 -11475.389,E2 -11475.389} C_VEL
LIN {X 0,Y 393.092,Z 460.576,A -85,B 0,C 180,E1 -11476.578,E2 -11476.578} C_VEL
LIN {X 0,Y 393.882,Z 450.453,A -85,B 0,C 180,E1 -11477.645,E2 -11477.645} C_VEL
LIN {X 0,Y 394.662,Z 439.43,A -85,B 0,C 180,E1 -11478.572,E2 -11478.572} C_VEL
LIN {X 0,Y 395.27,Z 428.765,A -85,B 0,C 180,E1 -11479.278,E2 -11479.278} C_VEL
LIN {X 0,Y 392.195,Z 415.526,A -85,B 0,C 180,E1 -11480.119,E2 -11480.119} C_VEL
LIN {X 0,Y 389.185,Z 405.333,A -85,B 0,C 180,E1 -11480.653,E2 -11480.653} C_VEL
LIN {X 0,Y 389.308,Z 401.868,A -85,B 0,C 180,E1 -11484.326,E2 -11484.326} C_VEL
LIN {X 0,Y 389.511,Z 398.477,A -85,B 0,C 180,E1 -11487.996,E2 -11487.996} C_VEL
LIN {X 0,Y 389.588,Z 395.904,A -85,B 0,C 180,E1 -11490.852,E2 -11490.852} C_VEL
LIN {X 0,Y 389.742,Z 392.758,A -85,B 0,C 180,E1 -11494.37,E2 -11494.37} C_VEL
LIN {X 0,Y 389.769,Z 391.937,A -85,B 0,C 180,E1 -11495.498,E2 -11495.498} C_VEL
LIN {X 0,Y 389.982,Z 391.914,A -85,B 0,C 180,E1 -11497.762,E2 -11497.762} C_VEL
LIN {X 0,Y 390.101,Z 391.896,A -85,B 0,C 180,E1 -11501.078,E2 -11501.078} C_VEL
LIN {X 0,Y 390.134,Z 391.89,A -85,B 0,C 180,E1 -11504.323,E2 -11504.323} C_VEL
LIN {X 0,Y 390.166,Z 391.886,A -85,B 0,C 180,E1 -11507.517,E2 -11507.517} C_VEL
LIN {X 0,Y 390.2,Z 391.881,A -85,B 0,C 180,E1 -11510.671,E2 -11510.671} C_VEL
LIN {X 0,Y 390.322,Z 391.866,A -85,B 0,C 180,E1 -11513.798,E2 -11513.798} C_VEL
LIN {X 0,Y 390.415,Z 391.854,A -85,B 0,C 180,E1 -11517.937,E2 -11517.937} C_VEL
LIN {X 0,Y 390.544,Z 391.836,A -85,B 0,C 180,E1 -11520,E2 -11520} C_VEL
LIN {X 0,Y 390.31,Z 391.868,A -85,B 0,C 180,E1 -11523.096,E2 -11523.096} C_VEL
LIN {X 0,Y 390.321,Z 391.866,A -85,B 0,C 180,E1 -11526.202,E2 -11526.202} C_VEL
LIN {X 0,Y 390.2,Z 391.881,A -85,B 0,C 180,E1 -11529.329,E2 -11529.329} C_VEL
LIN {X 0,Y 390.166,Z 391.885,A -85,B 0,C 180,E1 -11532.483,E2 -11532.483} C_VEL
LIN {X 0,Y 390.134,Z 391.888,A -85,B 0,C 180,E1 -11535.677,E2 -11535.677} C_VEL
LIN {X 0,Y 390.1,Z 391.89,A -85,B 0,C 180,E1 -11538.922,E2 -11538.922} C_VEL
LIN {X 0,Y 390.035,Z 391.903,A -85,B 0,C 180,E1 -11542.234,E2 -11542.234} C_VEL
LIN {X 0,Y 390.115,Z 391.892,A -85,B 0,C 180,E1 -11545.744,E2 -11545.744} C_VEL
LIN {X 0,Y 390.054,Z 391.898,A -85,B 0,C 180,E1 -11549.11,E2 -11549.11} C_VEL
LIN {X 0,Y 390.039,Z 391.904,A -85,B 0,C 180,E1 -11552.722,E2 -11552.722} C_VEL
LIN {X 0,Y 390.053,Z 391.904,A -85,B 0,C 180,E1 -11555.826,E2 -11555.826} C_VEL
LIN {X 0,Y 390.072,Z 391.9,A -85,B 0,C 180,E1 -11559.22,E2 -11559.22} C_VEL
LIN {X 0,Y 390.078,Z 391.898,A -85,B 0,C 180,E1 -11562.381,E2 -11562.381} C_VEL
LIN {X 0,Y 390.074,Z 391.988,A -85,B 0,C 180,E1 -11564.923,E2 -11564.923} C_VEL
LIN {X 0,Y 391.049,Z 397.259,A -85,B 0,C 180,E1 -11568.321,E2 -11568.321} C_VEL
LIN {X 0,Y 392.207,Z 403.68,A -85,B 0,C 180,E1 -11572.04,E2 -11572.04} C_VEL
LIN {X 0,Y 392.502,Z 406.931,A -85,B 0,C 180,E1 -11573.781,E2 -11573.781} C_VEL
LIN {X 0,Y 392.07,Z 411.903,A -85,B 0,C 180,E1 -11576.242,E2 -11576.242} C_VEL
LIN {X 0,Y 391.289,Z 419.456,A -85,B 0,C 180,E1 -11579.808,E2 -11579.808} C_VEL
LIN {X 0,Y 390.654,Z 427.122,A -85,B 0,C 180,E1 -11583.272,E2 -11583.272} C_VEL
LIN {X 0,Y 390.038,Z 436.34,A -85,B 0,C 180,E1 -11587.261,E2 -11587.261} C_VEL
LIN {X 0,Y 389.593,Z 445.345,A -85,B 0,C 180,E1 -11591.052,E2 -11591.052} C_VEL
LIN {X 0,Y 389.548,Z 446.122,A -85,B 0,C 180,E1 -11591.374,E2 -11591.374} C_VEL
LIN {X 0,Y 391.822,Z 459.809,A -85,B 0,C 180,E1 -11591.925,E2 -11591.925} C_VEL
LIN {X 0,Y 393.399,Z 472.276,A -85,B 0,C 180,E1 -11592.609,E2 -11592.609} C_VEL
LIN {X 0,Y 394.158,Z 479.314,A -85,B 0,C 180,E1 -11593.082,E2 -11593.082} C_VEL
LIN {X 0,Y 393.334,Z 490.701,A -85,B 0,C 180,E1 -11593.922,E2 -11593.922} C_VEL
LIN {X 0,Y 392.422,Z 501.684,A -85,B 0,C 180,E1 -11594.949,E2 -11594.949} C_VEL
LIN {X 0,Y 391.652,Z 511.387,A -85,B 0,C 180,E1 -11596.08,E2 -11596.08} C_VEL
LIN {X 0,Y 390.789,Z 521.519,A -85,B 0,C 180,E1 -11597.537,E2 -11597.537} C_VEL
LIN {X 0,Y 389.96,Z 530.215,A -85,B 0,C 180,E1 -11599.092,E2 -11599.092} C_VEL
LIN {X 0,Y 389.45,Z 537.188,A -85,B 0,C 180,E1 -11600.653,E2 -11600.653} C_VEL
LIN {X 0,Y 389.076,Z 542.787,A -85,B 0,C 180,E1 -11602.214,E2 -11602.214} C_VEL
LIN {X 0,Y 388.833,Z 547.975,A -85,B 0,C 180,E1 -11604.096,E2 -11604.096} C_VEL
LIN {X 0,Y 388.73,Z 551.423,A -85,B 0,C 180,E1 -11605.853,E2 -11605.853} C_VEL
LIN {X 0,Y 388.788,Z 553.877,A -85,B 0,C 180,E1 -11607.928,E2 -11607.928} C_VEL
LIN {X 0,Y 388.743,Z 554.503,A -85,B 0,C 180,E1 -11608.964,E2 -11608.964} C_VEL
LIN {X 0,Y 388.742,Z 554.73,A -85,B 0,C 180,E1 -11610,E2 -11610} C_VEL
LIN {X 0,Y 388.788,Z 553.915,A -85,B 0,C 180,E1 -11612.072,E2 -11612.072} C_VEL
LIN {X 0,Y 388.716,Z 552.91,A -85,B 0,C 180,E1 -11613.109,E2 -11613.109} C_VEL
LIN {X 0,Y 388.729,Z 551.499,A -85,B 0,C 180,E1 -11614.147,E2 -11614.147} C_VEL
LIN {X 0,Y 388.83,Z 548.081,A -85,B 0,C 180,E1 -11615.9,E2 -11615.9} C_VEL
LIN {X 0,Y 389.077,Z 542.914,A -85,B 0,C 180,E1 -11617.786,E2 -11617.786} C_VEL
LIN {X 0,Y 389.452,Z 537.336,A -85,B 0,C 180,E1 -11619.347,E2 -11619.347} C_VEL
LIN {X 0,Y 389.956,Z 530.374,A -85,B 0,C 180,E1 -11620.908,E2 -11620.908} C_VEL
LIN {X 0,Y 390.799,Z 521.663,A -85,B 0,C 180,E1 -11622.462,E2 -11622.462} C_VEL
LIN {X 0,Y 391.544,Z 512.988,A -85,B 0,C 180,E1 -11623.724,E2 -11623.724} C_VEL
LIN {X 0,Y 392.321,Z 502.947,A -85,B 0,C 180,E1 -11624.922,E2 -11624.922} C_VEL
LIN {X 0,Y 393.184,Z 492.237,A -85,B 0,C 180,E1 -11625.951,E2 -11625.951} C_VEL
LIN {X 0,Y 394.054,Z 480.909,A -85,B 0,C 180,E1 -11626.803,E2 -11626.803} C_VEL
LIN {X 0,Y 393.833,Z 475.744,A -85,B 0,C 180,E1 -11627.148,E2 -11627.148} C_VEL
LIN {X 0,Y 392.036,Z 462.144,A -85,B 0,C 180,E1 -11627.929,E2 -11627.929} C_VEL
LIN {X 0,Y 389.964,Z 449.292,A -85,B 0,C 180,E1 -11628.47,E2 -11628.47} C_VEL
LIN {X 0,Y 389.564,Z 446.768,A -85,B 0,C 180,E1 -11628.573,E2 -11628.573} C_VEL
LIN {X 0,Y 389.958,Z 439.385,A -85,B 0,C 180,E1 -11631.682,E2 -11631.682} C_VEL
LIN {X 0,Y 390.437,Z 431.582,A -85,B 0,C 180,E1 -11635.024,E2 -11635.024} C_VEL
LIN {X 0,Y 390.988,Z 424.208,A -85,B 0,C 180,E1 -11638.264,E2 -11638.264} C_VEL
LIN {X 0,Y 391.728,Z 416.117,A -85,B 0,C 180,E1 -11641.946,E2 -11641.946} C_VEL
LIN {X 0,Y 392.486,Z 408.408,A -85,B 0,C 180,E1 -11645.587,E2 -11645.587} C_VEL
LIN {X 0,Y 392.345,Z 404.571,A -85,B 0,C 180,E1 -11647.519,E2 -11647.519} C_VEL
LIN {X 0,Y 391.452,Z 399.43,A -85,B 0,C 180,E1 -11650.264,E2 -11650.264} C_VEL
LIN {X 0,Y 390.251,Z 393.036,A -85,B 0,C 180,E1 -11653.916,E2 -11653.916} C_VEL
LIN {X 0,Y 390.051,Z 391.901,A -85,B 0,C 180,E1 -11654.643,E2 -11654.643} C_VEL
LIN {X 0,Y 390.063,Z 391.899,A -85,B 0,C 180,E1 -11658.191,E2 -11658.191} C_VEL
LIN {X 0,Y 390.09,Z 391.897,A -85,B 0,C 180,E1 -11660.908,E2 -11660.908} C_VEL
LIN {X 0,Y 390.08,Z 391.897,A -85,B 0,C 180,E1 -11664.792,E2 -11664.792} C_VEL
LIN {X 0,Y 390.017,Z 391.903,A -85,B 0,C 180,E1 -11668.495,E2 -11668.495} C_VEL
LIN {X 0,Y 390.11,Z 391.89,A -85,B 0,C 180,E1 -11672.069,E2 -11672.069} C_VEL
LIN {X 0,Y 390.072,Z 391.895,A -85,B 0,C 180,E1 -11675.519,E2 -11675.519} C_VEL
LIN {X 0,Y 390.048,Z 391.901,A -85,B 0,C 180,E1 -11678.877,E2 -11678.877} C_VEL
LIN {X 0,Y 390.12,Z 391.889,A -85,B 0,C 180,E1 -11682.166,E2 -11682.166} C_VEL
LIN {X 0,Y 390.135,Z 391.887,A -85,B 0,C 180,E1 -11685.392,E2 -11685.392} C_VEL
LIN {X 0,Y 390.141,Z 391.89,A -85,B 0,C 180,E1 -11688.571,E2 -11688.571} C_VEL
LIN {X 0,Y 390.299,Z 391.867,A -85,B 0,C 180,E1 -11692.031,E2 -11692.031} C_VEL
LIN {X 0,Y 390.219,Z 391.88,A -85,B 0,C 180,E1 -11694.833,E2 -11694.833} C_VEL
LIN {X 0,Y 390.412,Z 391.852,A -85,B 0,C 180,E1 -11697.937,E2 -11697.937} C_VEL
LIN {X 0,Y 390.543,Z 391.836,A -85,B 0,C 180,E1 -11700,E2 -11700} C_VEL
LIN {X 0,Y 390.308,Z 391.866,A -85,B 0,C 180,E1 -11703.097,E2 -11703.097} C_VEL
LIN {X 0,Y 390.301,Z 391.865,A -85,B 0,C 180,E1 -11706.637,E2 -11706.637} C_VEL
LIN {X 0,Y 390.197,Z 391.879,A -85,B 0,C 180,E1 -11709.329,E2 -11709.329} C_VEL
LIN {X 0,Y 390.186,Z 391.88,A -85,B 0,C 180,E1 -11713.439,E2 -11713.439} C_VEL
LIN {X 0,Y 390.141,Z 391.885,A -85,B 0,C 180,E1 -11717.308,E2 -11717.308} C_VEL
LIN {X 0,Y 390.08,Z 391.898,A -85,B 0,C 180,E1 -11720.471,E2 -11720.471} C_VEL
LIN {X 0,Y 390.082,Z 391.893,A -85,B 0,C 180,E1 -11723.352,E2 -11723.352} C_VEL
LIN {X 0,Y 390.107,Z 391.892,A -85,B 0,C 180,E1 -11726.769,E2 -11726.769} C_VEL
LIN {X 0,Y 390.033,Z 391.904,A -85,B 0,C 180,E1 -11730.301,E2 -11730.301} C_VEL
LIN {X 0,Y 390.063,Z 391.899,A -85,B 0,C 180,E1 -11734.026,E2 -11734.026} C_VEL
LIN {X 0,Y 390.043,Z 391.898,A -85,B 0,C 180,E1 -11737.553,E2 -11737.553} C_VEL
LIN {X 0,Y 390.073,Z 391.895,A -85,B 0,C 180,E1 -11740.826,E2 -11740.826} C_VEL
LIN {X 0,Y 390.052,Z 391.9,A -85,B 0,C 180,E1 -11743.887,E2 -11743.887} C_VEL
LIN {X 0,Y 390.054,Z 391.897,A -85,B 0,C 180,E1 -11746.791,E2 -11746.791} C_VEL
LIN {X 0,Y 390.055,Z 391.898,A -85,B 0,C 180,E1 -11749.562,E2 -11749.562} C_VEL
LIN {X 0,Y 390.044,Z 391.9,A -85,B 0,C 180,E1 -11752.45,E2 -11752.45} C_VEL
LIN {X 0,Y 390.083,Z 391.897,A -85,B 0,C 180,E1 -11756.048,E2 -11756.048} C_VEL
LIN {X 0,Y 390.046,Z 391.901,A -85,B 0,C 180,E1 -11759.87,E2 -11759.87} C_VEL
LIN {X 0,Y 390.114,Z 391.889,A -85,B 0,C 180,E1 -11763.233,E2 -11763.233} C_VEL
LIN {X 0,Y 390.108,Z 391.89,A -85,B 0,C 180,E1 -11766.751,E2 -11766.751} C_VEL
LIN {X 0,Y 390.106,Z 391.895,A -85,B 0,C 180,E1 -11769.984,E2 -11769.984} C_VEL
LIN {X 0,Y 390.14,Z 391.886,A -85,B 0,C 180,E1 -11773.249,E2 -11773.249} C_VEL
LIN {X 0,Y 390.197,Z 391.879,A -85,B 0,C 180,E1 -11776.562,E2 -11776.562} C_VEL
LIN {X 0,Y 390.208,Z 391.877,A -85,B 0,C 180,E1 -11780.672,E2 -11780.672} C_VEL
LIN {X 0,Y 390.322,Z 391.863,A -85,B 0,C 180,E1 -11782.76,E2 -11782.76} C_VEL
LIN {X 0,Y 390.228,Z 391.875,A -85,B 0,C 180,E1 -11784.834,E2 -11784.834} C_VEL
LIN {X 0,Y 390.336,Z 391.866,A -85,B 0,C 180,E1 -11787.937,E2 -11787.937} C_VEL
LIN {X 0,Y 390.038,Z 391.903,A -85,B 0,C 180,E1 -11790,E2 -11790} C_VEL
LIN {X 0,Y 389.537,Z 391.967,A -85,B 0,C 180,E1 -11791.034,E2 -11791.034} C_VEL
LIN {X 0,Y 389.614,Z 394.627,A -85,B 0,C 180,E1 -11794.138,E2 -11794.138} C_VEL
LIN {X 0,Y 389.454,Z 397.643,A -85,B 0,C 180,E1 -11797.257,E2 -11797.257} C_VEL
LIN {X 0,Y 389.263,Z 400.735,A -85,B 0,C 180,E1 -11800.402,E2 -11800.402} C_VEL
LIN {X 0,Y 389.204,Z 404.041,A -85,B 0,C 180,E1 -11803.643,E2 -11803.643} C_VEL
LIN {X 0,Y 392.84,Z 418.394,A -85,B 0,C 180,E1 -11804.372,E2 -11804.372} C_VEL
LIN {X 0,Y 394.911,Z 427.773,A -85,B 0,C 180,E1 -11804.967,E2 -11804.967} C_VEL
LIN {X 0,Y 394.2,Z 440.225,A -85,B 0,C 180,E1 -11805.795,E2 -11805.795} C_VEL
LIN {X 0,Y 393.49,Z 451.092,A -85,B 0,C 180,E1 -11806.738,E2 -11806.738} C_VEL
LIN {X 0,Y 392.654,Z 461.683,A -85,B 0,C 180,E1 -11807.888,E2 -11807.888} C_VEL
LIN {X 0,Y 391.849,Z 470.822,A -85,B 0,C 180,E1 -11809.106,E2 -11809.106} C_VEL
LIN {X 0,Y 391.086,Z 479.049,A -85,B 0,C 180,E1 -11810.443,E2 -11810.443} C_VEL
LIN {X 0,Y 390.405,Z 486.516,A -85,B 0,C 180,E1 -11811.934,E2 -11811.934} C_VEL
LIN {X 0,Y 390.196,Z 488.815,A -85,B 0,C 180,E1 -11812.467,E2 -11812.467} C_VEL
LIN {X 0,Y 389.296,Z 491.828,A -85,B 0,C 180,E1 -11813.206,E2 -11813.206} C_VEL
LIN {X 0,Y 386.092,Z 496.29,A -85,B 0,C 180,E1 -11814.425,E2 -11814.425} C_VEL
LIN {X 0,Y 382.951,Z 500.125,A -85,B 0,C 180,E1 -11815.708,E2 -11815.708} C_VEL
LIN {X 0,Y 382.161,Z 502.032,A -85,B 0,C 180,E1 -11816.538,E2 -11816.538} C_VEL
LIN {X 0,Y 381.889,Z 504.622,A -85,B 0,C 180,E1 -11817.949,E2 -11817.949} C_VEL
LIN {X 0,Y 381.663,Z 507.014,A -85,B 0,C 180,E1 -11820.063,E2 -11820.063} C_VEL
LIN {X 0,Y 381.614,Z 507.845,A -85,B 0,C 180,E1 -11822.095,E2 -11822.095} C_VEL
LIN {X 0,Y 381.691,Z 507.22,A -85,B 0,C 180,E1 -11824.047,E2 -11824.047} C_VEL
LIN {X 0,Y 381.918,Z 505.143,A -85,B 0,C 180,E1 -11826.076,E2 -11826.076} C_VEL
LIN {X 0,Y 382.216,Z 502.267,A -85,B 0,C 180,E1 -11827.752,E2 -11827.752} C_VEL
LIN {X 0,Y 382.645,Z 498.013,A -85,B 0,C 180,E1 -11829.519,E2 -11829.519} C_VEL
LIN {X 0,Y 383.187,Z 492.176,A -85,B 0,C 180,E1 -11831.32,E2 -11831.32} C_VEL
LIN {X 0,Y 383.949,Z 484.649,A -85,B 0,C 180,E1 -11833.117,E2 -11833.117} C_VEL
LIN {X 0,Y 384.781,Z 476.393,A -85,B 0,C 180,E1 -11834.671,E2 -11834.671} C_VEL
LIN {X 0,Y 385.774,Z 466.27,A -85,B 0,C 180,E1 -11836.189,E2 -11836.189} C_VEL
LIN {X 0,Y 386.674,Z 456.211,A -85,B 0,C 180,E1 -11837.4,E2 -11837.4} C_VEL
LIN {X 0,Y 387.578,Z 444.505,A -85,B 0,C 180,E1 -11838.514,E2 -11838.514} C_VEL
LIN {X 0,Y 388.378,Z 433.25,A -85,B 0,C 180,E1 -11839.349,E2 -11839.349} C_VEL
LIN {X 0,Y 388.491,Z 429.887,A -85,B 0,C 180,E1 -11839.563,E2 -11839.563} C_VEL
LIN {X 0,Y 385.477,Z 417.023,A -85,B 0,C 180,E1 -11840.417,E2 -11840.417} C_VEL
LIN {X 0,Y 382.15,Z 405.805,A -85,B 0,C 180,E1 -11841.018,E2 -11841.018} C_VEL
LIN {X 0,Y 382.238,Z 403.032,A -85,B 0,C 180,E1 -11843.998,E2 -11843.998} C_VEL
LIN {X 0,Y 382.46,Z 399.551,A -85,B 0,C 180,E1 -11847.798,E2 -11847.798} C_VEL
LIN {X 0,Y 382.577,Z 396.295,A -85,B 0,C 180,E1 -11851.469,E2 -11851.469} C_VEL
LIN {X 0,Y 382.696,Z 393.191,A -85,B 0,C 180,E1 -11855.015,E2 -11855.015} C_VEL
LIN {X 0,Y 382.873,Z 392.799,A -85,B 0,C 180,E1 -11856.604,E2 -11856.604} C_VEL
LIN {X 0,Y 383.05,Z 392.776,A -85,B 0,C 180,E1 -11859.598,E2 -11859.598} C_VEL
LIN {X 0,Y 383.1,Z 392.765,A -85,B 0,C 180,E1 -11862.931,E2 -11862.931} C_VEL
LIN {X 0,Y 383.121,Z 392.764,A -85,B 0,C 180,E1 -11866.464,E2 -11866.464} C_VEL
LIN {X 0,Y 383.147,Z 392.759,A -85,B 0,C 180,E1 -11870.498,E2 -11870.498} C_VEL
LIN {X 0,Y 383.278,Z 392.744,A -85,B 0,C 180,E1 -11873.683,E2 -11873.683} C_VEL
LIN {X 0,Y 383.382,Z 392.73,A -85,B 0,C 180,E1 -11877.899,E2 -11877.899} C_VEL
LIN {X 0,Y 383.514,Z 392.711,A -85,B 0,C 180,E1 -11880,E2 -11880} C_VEL
LIN {X 0,Y 383.246,Z 392.747,A -85,B 0,C 180,E1 -11883.154,E2 -11883.154} C_VEL
LIN {X 0,Y 383.277,Z 392.745,A -85,B 0,C 180,E1 -11886.316,E2 -11886.316} C_VEL
LIN {X 0,Y 383.147,Z 392.76,A -85,B 0,C 180,E1 -11889.502,E2 -11889.502} C_VEL
LIN {X 0,Y 383.12,Z 392.76,A -85,B 0,C 180,E1 -11893.536,E2 -11893.536} C_VEL
LIN {X 0,Y 383.09,Z 392.767,A -85,B 0,C 180,E1 -11897.455,E2 -11897.455} C_VEL
LIN {X 0,Y 383.024,Z 392.776,A -85,B 0,C 180,E1 -11900.647,E2 -11900.647} C_VEL
LIN {X 0,Y 383.029,Z 392.775,A -85,B 0,C 180,E1 -11903.808,E2 -11903.808} C_VEL
LIN {X 0,Y 383.076,Z 392.767,A -85,B 0,C 180,E1 -11906.124,E2 -11906.124} C_VEL
LIN {X 0,Y 382.988,Z 392.782,A -85,B 0,C 180,E1 -11909.7,E2 -11909.7} C_VEL
LIN {X 0,Y 382.999,Z 392.78,A -85,B 0,C 180,E1 -11913.401,E2 -11913.401} C_VEL
LIN {X 0,Y 383.03,Z 392.779,A -85,B 0,C 180,E1 -11916.165,E2 -11916.165} C_VEL
LIN {X 0,Y 383.017,Z 392.778,A -85,B 0,C 180,E1 -11919.957,E2 -11919.957} C_VEL
LIN {X 0,Y 383.03,Z 392.774,A -85,B 0,C 180,E1 -11922.783,E2 -11922.783} C_VEL
LIN {X 0,Y 383.018,Z 392.78,A -85,B 0,C 180,E1 -11924.399,E2 -11924.399} C_VEL
LIN {X 0,Y 383.833,Z 397.192,A -85,B 0,C 180,E1 -11927.354,E2 -11927.354} C_VEL
LIN {X 0,Y 384.655,Z 401.919,A -85,B 0,C 180,E1 -11930.247,E2 -11930.247} C_VEL
LIN {X 0,Y 385.478,Z 406.746,A -85,B 0,C 180,E1 -11933.012,E2 -11933.012} C_VEL
LIN {X 0,Y 385.302,Z 410.887,A -85,B 0,C 180,E1 -11935.166,E2 -11935.166} C_VEL
LIN {X 0,Y 384.489,Z 417.938,A -85,B 0,C 180,E1 -11938.605,E2 -11938.605} C_VEL
LIN {X 0,Y 383.802,Z 425.532,A -85,B 0,C 180,E1 -11942.164,E2 -11942.164} C_VEL
LIN {X 0,Y 383.19,Z 433.24,A -85,B 0,C 180,E1 -11945.628,E2 -11945.628} C_VEL
LIN {X 0,Y 382.676,Z 442.153,A -85,B 0,C 180,E1 -11949.495,E2 -11949.495} C_VEL
LIN {X 0,Y 382.534,Z 445.674,A -85,B 0,C 180,E1 -11951.003,E2 -11951.003} C_VEL
LIN {X 0,Y 384.824,Z 459.312,A -85,B 0,C 180,E1 -11951.568,E2 -11951.568} C_VEL
LIN {X 0,Y 386.434,Z 472.485,A -85,B 0,C 180,E1 -11952.316,E2 -11952.316} C_VEL
LIN {X 0,Y 387.251,Z 480.822,A -85,B 0,C 180,E1 -11952.897,E2 -11952.897} C_VEL
LIN {X 0,Y 386.209,Z 493.298,A -85,B 0,C 180,E1 -11953.888,E2 -11953.888} C_VEL
LIN {X 0,Y 385.173,Z 504.844,A -85,B 0,C 180,E1 -11955.065,E2 -11955.065} C_VEL
LIN {X 0,Y 384.426,Z 514.181,A -85,B 0,C 180,E1 -11956.251,E2 -11956.251} C_VEL
LIN {X 0,Y 383.64,Z 522.711,A -85,B 0,C 180,E1 -11957.57,E2 -11957.57} C_VEL
LIN {X 0,Y 382.837,Z 531.054,A -85,B 0,C 180,E1 -11959.154,E2 -11959.154} C_VEL
LIN {X 0,Y 382.332,Z 537.8,A -85,B 0,C 180,E1 -11960.744,E2 -11960.744} C_VEL
LIN {X 0,Y 381.926,Z 543.983,A -85,B 0,C 180,E1 -11962.599,E2 -11962.599} C_VEL
LIN {X 0,Y 381.733,Z 547.922,A -85,B 0,C 180,E1 -11964.145,E2 -11964.145} C_VEL
LIN {X 0,Y 381.658,Z 551,A -85,B 0,C 180,E1 -11965.776,E2 -11965.776} C_VEL
LIN {X 0,Y 381.704,Z 553.449,A -85,B 0,C 180,E1 -11967.889,E2 -11967.889} C_VEL
LIN {X 0,Y 381.676,Z 554.076,A -85,B 0,C 180,E1 -11968.945,E2 -11968.945} C_VEL
LIN {X 0,Y 381.672,Z 554.301,A -85,B 0,C 180,E1 -11970,E2 -11970} C_VEL
LIN {X 0,Y 381.676,Z 554.088,A -85,B 0,C 180,E1 -11971.055,E2 -11971.055} C_VEL
LIN {X 0,Y 381.704,Z 553.482,A -85,B 0,C 180,E1 -11972.11,E2 -11972.11} C_VEL
LIN {X 0,Y 381.657,Z 551.061,A -85,B 0,C 180,E1 -11974.224,E2 -11974.224} C_VEL
LIN {X 0,Y 381.732,Z 548.005,A -85,B 0,C 180,E1 -11975.852,E2 -11975.852} C_VEL
LIN {X 0,Y 381.927,Z 544.075,A -85,B 0,C 180,E1 -11977.4,E2 -11977.4} C_VEL
LIN {X 0,Y 382.333,Z 537.889,A -85,B 0,C 180,E1 -11979.255,E2 -11979.255} C_VEL
LIN {X 0,Y 382.834,Z 531.141,A -85,B 0,C 180,E1 -11980.845,E2 -11980.845} C_VEL
LIN {X 0,Y 383.649,Z 522.785,A -85,B 0,C 180,E1 -11982.429,E2 -11982.429} C_VEL
LIN {X 0,Y 384.444,Z 514.195,A -85,B 0,C 180,E1 -11983.747,E2 -11983.747} C_VEL
LIN {X 0,Y 385.321,Z 503.604,A -85,B 0,C 180,E1 -11985.064,E2 -11985.064} C_VEL
LIN {X 0,Y 386.202,Z 493.138,A -85,B 0,C 180,E1 -11986.111,E2 -11986.111} C_VEL
LIN {X 0,Y 387.125,Z 482.049,A -85,B 0,C 180,E1 -11986.992,E2 -11986.992} C_VEL
LIN {X 0,Y 387.033,Z 477.375,A -85,B 0,C 180,E1 -11987.318,E2 -11987.318} C_VEL
LIN {X 0,Y 385.364,Z 464.169,A -85,B 0,C 180,E1 -11988.129,E2 -11988.129} C_VEL
LIN {X 0,Y 383.135,Z 450.213,A -85,B 0,C 180,E1 -11988.761,E2 -11988.761} C_VEL
LIN {X 0,Y 382.518,Z 446.44,A -85,B 0,C 180,E1 -11988.89,E2 -11988.89} C_VEL
LIN {X 0,Y 382.916,Z 438.994,A -85,B 0,C 180,E1 -11992.101,E2 -11992.101} C_VEL
LIN {X 0,Y 383.469,Z 431.223,A -85,B 0,C 180,E1 -11995.511,E2 -11995.511} C_VEL
LIN {X 0,Y 384.111,Z 423.473,A -85,B 0,C 180,E1 -11999.01,E2 -11999.01} C_VEL
LIN {X 0,Y 384.845,Z 415.262,A -85,B 0,C 180,E1 -12002.855,E2 -12002.855} C_VEL
LIN {X 0,Y 385.479,Z 409.379,A -85,B 0,C 180,E1 -12005.69,E2 -12005.69} C_VEL
LIN {X 0,Y 385.342,Z 405.596,A -85,B 0,C 180,E1 -12007.642,E2 -12007.642} C_VEL
LIN {X 0,Y 384.403,Z 400.418,A -85,B 0,C 180,E1 -12010.472,E2 -12010.472} C_VEL
LIN {X 0,Y 383.418,Z 395.029,A -85,B 0,C 180,E1 -12013.592,E2 -12013.592} C_VEL
LIN {X 0,Y 383.016,Z 392.778,A -85,B 0,C 180,E1 -12015.05,E2 -12015.05} C_VEL
LIN {X 0,Y 383.035,Z 392.775,A -85,B 0,C 180,E1 -12017.243,E2 -12017.243} C_VEL
LIN {X 0,Y 383.017,Z 392.776,A -85,B 0,C 180,E1 -12020.411,E2 -12020.411} C_VEL
LIN {X 0,Y 383.021,Z 392.772,A -85,B 0,C 180,E1 -12024.044,E2 -12024.044} C_VEL
LIN {X 0,Y 382.98,Z 392.778,A -85,B 0,C 180,E1 -12027.577,E2 -12027.577} C_VEL
LIN {X 0,Y 382.985,Z 392.777,A -85,B 0,C 180,E1 -12030.299,E2 -12030.299} C_VEL
LIN {X 0,Y 383.073,Z 392.766,A -85,B 0,C 180,E1 -12034.02,E2 -12034.02} C_VEL
LIN {X 0,Y 383,Z 392.776,A -85,B 0,C 180,E1 -12037.335,E2 -12037.335} C_VEL
LIN {X 0,Y 383.052,Z 392.773,A -85,B 0,C 180,E1 -12040.716,E2 -12040.716} C_VEL
LIN {X 0,Y 383.072,Z 392.766,A -85,B 0,C 180,E1 -12044.026,E2 -12044.026} C_VEL
LIN {X 0,Y 383.128,Z 392.76,A -85,B 0,C 180,E1 -12047.284,E2 -12047.284} C_VEL
LIN {X 0,Y 383.143,Z 392.761,A -85,B 0,C 180,E1 -12050.498,E2 -12050.498} C_VEL
LIN {X 0,Y 383.274,Z 392.741,A -85,B 0,C 180,E1 -12053.684,E2 -12053.684} C_VEL
LIN {X 0,Y 383.379,Z 392.728,A -85,B 0,C 180,E1 -12057.899,E2 -12057.899} C_VEL
LIN {X 0,Y 383.513,Z 392.712,A -85,B 0,C 180,E1 -12060,E2 -12060} C_VEL
LIN {X 0,Y 383.244,Z 392.746,A -85,B 0,C 180,E1 -12063.154,E2 -12063.154} C_VEL
LIN {X 0,Y 383.261,Z 392.743,A -85,B 0,C 180,E1 -12066.632,E2 -12066.632} C_VEL
LIN {X 0,Y 383.252,Z 392.748,A -85,B 0,C 180,E1 -12068.436,E2 -12068.436} C_VEL
LIN {X 0,Y 383.09,Z 392.764,A -85,B 0,C 180,E1 -12071.642,E2 -12071.642} C_VEL
LIN {X 0,Y 383.102,Z 392.764,A -85,B 0,C 180,E1 -12074.882,E2 -12074.882} C_VEL
LIN {X 0,Y 383.081,Z 392.768,A -85,B 0,C 180,E1 -12078.173,E2 -12078.173} C_VEL
LIN {X 0,Y 382.986,Z 392.777,A -85,B 0,C 180,E1 -12081.532,E2 -12081.532} C_VEL
LIN {X 0,Y 383.046,Z 392.77,A -85,B 0,C 180,E1 -12084.961,E2 -12084.961} C_VEL
LIN {X 0,Y 383.034,Z 392.775,A -85,B 0,C 180,E1 -12088.493,E2 -12088.493} C_VEL
LIN {X 0,Y 383.004,Z 392.779,A -85,B 0,C 180,E1 -12092.151,E2 -12092.151} C_VEL
LIN {X 0,Y 383.013,Z 392.775,A -85,B 0,C 180,E1 -12094.669,E2 -12094.669} C_VEL
LIN {X 0,Y 382.999,Z 392.778,A -85,B 0,C 180,E1 -12097.905,E2 -12097.905} C_VEL
LIN {X 0,Y 383.009,Z 392.774,A -85,B 0,C 180,E1 -12101.344,E2 -12101.344} C_VEL
LIN {X 0,Y 382.993,Z 392.78,A -85,B 0,C 180,E1 -12104.304,E2 -12104.304} C_VEL
LIN {X 0,Y 383.007,Z 392.774,A -85,B 0,C 180,E1 -12107.241,E2 -12107.241} C_VEL
LIN {X 0,Y 383.014,Z 392.776,A -85,B 0,C 180,E1 -12110.414,E2 -12110.414} C_VEL
LIN {X 0,Y 383.025,Z 392.776,A -85,B 0,C 180,E1 -12114.046,E2 -12114.046} C_VEL
LIN {X 0,Y 382.986,Z 392.779,A -85,B 0,C 180,E1 -12117.579,E2 -12117.579} C_VEL
LIN {X 0,Y 382.992,Z 392.779,A -85,B 0,C 180,E1 -12120.301,E2 -12120.301} C_VEL
LIN {X 0,Y 383.081,Z 392.769,A -85,B 0,C 180,E1 -12124.022,E2 -12124.022} C_VEL
LIN {X 0,Y 383.01,Z 392.775,A -85,B 0,C 180,E1 -12127.336,E2 -12127.336} C_VEL
LIN {X 0,Y 383.062,Z 392.767,A -85,B 0,C 180,E1 -12130.717,E2 -12130.717} C_VEL
LIN {X 0,Y 383.084,Z 392.769,A -85,B 0,C 180,E1 -12134.027,E2 -12134.027} C_VEL
LIN {X 0,Y 383.139,Z 392.759,A -85,B 0,C 180,E1 -12137.285,E2 -12137.285} C_VEL
LIN {X 0,Y 383.154,Z 392.756,A -85,B 0,C 180,E1 -12140.498,E2 -12140.498} C_VEL
LIN {X 0,Y 383.277,Z 392.74,A -85,B 0,C 180,E1 -12142.626,E2 -12142.626} C_VEL
LIN {X 0,Y 383.201,Z 392.75,A -85,B 0,C 180,E1 -12144.739,E2 -12144.739} C_VEL
LIN {X 0,Y 383.301,Z 392.743,A -85,B 0,C 180,E1 -12147.899,E2 -12147.899} C_VEL
LIN {X 0,Y 382.978,Z 392.782,A -85,B 0,C 180,E1 -12150,E2 -12150} C_VEL
LIN {X 0,Y 382.481,Z 392.846,A -85,B 0,C 180,E1 -12151.053,E2 -12151.053} C_VEL
LIN {X 0,Y 382.575,Z 395.524,A -85,B 0,C 180,E1 -12154.214,E2 -12154.214} C_VEL
LIN {X 0,Y 382.399,Z 398.605,A -85,B 0,C 180,E1 -12157.392,E2 -12157.392} C_VEL
LIN {X 0,Y 382.19,Z 401.712,A -85,B 0,C 180,E1 -12160.596,E2 -12160.596} C_VEL
LIN {X 0,Y 382.14,Z 404.414,A -85,B 0,C 180,E1 -12163.324,E2 -12163.324} C_VEL
LIN {X 0,Y 385.88,Z 418.898,A -85,B 0,C 180,E1 -12164.066,E2 -12164.066} C_VEL
LIN {X 0,Y 388.079,Z 429.665,A -85,B 0,C 180,E1 -12164.765,E2 -12164.765} C_VEL
LIN {X 0,Y 387.324,Z 441.28,A -85,B 0,C 180,E1 -12165.57,E2 -12165.57} C_VEL
LIN {X 0,Y 386.486,Z 452.868,A -85,B 0,C 180,E1 -12166.615,E2 -12166.615} C_VEL
LIN {X 0,Y 385.641,Z 463.132,A -85,B 0,C 180,E1 -12167.773,E2 -12167.773} C_VEL
LIN {X 0,Y 384.888,Z 471.794,A -85,B 0,C 180,E1 -12168.97,E2 -12168.97} C_VEL
LIN {X 0,Y 384.079,Z 480.004,A -85,B 0,C 180,E1 -12170.345,E2 -12170.345} C_VEL
LIN {X 0,Y 383.401,Z 487.042,A -85,B 0,C 180,E1 -12171.789,E2 -12171.789} C_VEL
LIN {X 0,Y 382.843,Z 493.303,A -85,B 0,C 180,E1 -12173.383,E2 -12173.383} C_VEL
LIN {X 0,Y 382.385,Z 498.36,A -85,B 0,C 180,E1 -12175.007,E2 -12175.007} C_VEL
LIN {X 0,Y 382.161,Z 502.032,A -85,B 0,C 180,E1 -12176.538,E2 -12176.538} C_VEL
LIN {X 0,Y 381.376,Z 503.722,A -85,B 0,C 180,E1 -12177.379,E2 -12177.379} C_VEL
LIN {X 0,Y 378.29,Z 505.982,A -85,B 0,C 180,E1 -12178.759,E2 -12178.759} C_VEL
LIN {X 0,Y 375.717,Z 507.258,A -85,B 0,C 180,E1 -12179.89,E2 -12179.89} C_VEL
LIN {X 0,Y 374.607,Z 507.897,A -85,B 0,C 180,E1 -12180.776,E2 -12180.776} C_VEL
LIN {X 0,Y 374.513,Z 507.978,A -85,B 0,C 180,E1 -12181.078,E2 -12181.078} C_VEL
LIN {X 0,Y 374.534,Z 508.187,A -85,B 0,C 180,E1 -12182.968,E2 -12182.968} C_VEL
LIN {X 0,Y 374.62,Z 507.471,A -85,B 0,C 180,E1 -12184.365,E2 -12184.365} C_VEL
LIN {X 0,Y 374.866,Z 505.439,A -85,B 0,C 180,E1 -12186.276,E2 -12186.276} C_VEL
LIN {X 0,Y 375.234,Z 502.097,A -85,B 0,C 180,E1 -12188.175,E2 -12188.175} C_VEL
LIN {X 0,Y 375.672,Z 497.77,A -85,B 0,C 180,E1 -12189.912,E2 -12189.912} C_VEL
LIN {X 0,Y 376.246,Z 492.085,A -85,B 0,C 180,E1 -12191.654,E2 -12191.654} C_VEL
LIN {X 0,Y 377.034,Z 484.967,A -85,B 0,C 180,E1 -12193.367,E2 -12193.367} C_VEL
LIN {X 0,Y 377.929,Z 476.592,A -85,B 0,C 180,E1 -12194.962,E2 -12194.962} C_VEL
LIN {X 0,Y 378.856,Z 467.622,A -85,B 0,C 180,E1 -12196.341,E2 -12196.341} C_VEL
LIN {X 0,Y 379.77,Z 457.646,A -85,B 0,C 180,E1 -12197.589,E2 -12197.589} C_VEL
LIN {X 0,Y 380.619,Z 447.523,A -85,B 0,C 180,E1 -12198.612,E2 -12198.612} C_VEL
LIN {X 0,Y 381.512,Z 436.1,A -85,B 0,C 180,E1 -12199.518,E2 -12199.518} C_VEL
LIN {X 0,Y 381.673,Z 430.847,A -85,B 0,C 180,E1 -12199.873,E2 -12199.873} C_VEL
LIN {X 0,Y 378.64,Z 418.14,A -85,B 0,C 180,E1 -12200.749,E2 -12200.749} C_VEL
LIN {X 0,Y 375.084,Z 406.264,A -85,B 0,C 180,E1 -12201.421,E2 -12201.421} C_VEL
LIN {X 0,Y 375.187,Z 403.444,A -85,B 0,C 180,E1 -12204.5,E2 -12204.5} C_VEL
LIN {X 0,Y 375.379,Z 400.816,A -85,B 0,C 180,E1 -12207.405,E2 -12207.405} C_VEL
LIN {X 0,Y 375.515,Z 397.742,A -85,B 0,C 180,E1 -12210.882,E2 -12210.882} C_VEL
LIN {X 0,Y 375.646,Z 394.61,A -85,B 0,C 180,E1 -12214.513,E2 -12214.513} C_VEL
LIN {X 0,Y 375.701,Z 393.69,A -85,B 0,C 180,E1 -12215.698,E2 -12215.698} C_VEL
LIN {X 0,Y 375.891,Z 393.669,A -85,B 0,C 180,E1 -12218.041,E2 -12218.041} C_VEL
LIN {X 0,Y 376.004,Z 393.65,A -85,B 0,C 180,E1 -12221.473,E2 -12221.473} C_VEL
LIN {X 0,Y 376.053,Z 393.645,A -85,B 0,C 180,E1 -12224.832,E2 -12224.832} C_VEL
LIN {X 0,Y 376.046,Z 393.645,A -85,B 0,C 180,E1 -12228.136,E2 -12228.136} C_VEL
LIN {X 0,Y 376.214,Z 393.623,A -85,B 0,C 180,E1 -12231.918,E2 -12231.918} C_VEL
LIN {X 0,Y 376.166,Z 393.627,A -85,B 0,C 180,E1 -12234.64,E2 -12234.64} C_VEL
LIN {X 0,Y 376.348,Z 393.606,A -85,B 0,C 180,E1 -12237.859,E2 -12237.859} C_VEL
LIN {X 0,Y 376.483,Z 393.587,A -85,B 0,C 180,E1 -12240,E2 -12240} C_VEL
LIN {X 0,Y 376.184,Z 393.627,A -85,B 0,C 180,E1 -12243.213,E2 -12243.213} C_VEL
LIN {X 0,Y 376.236,Z 393.623,A -85,B 0,C 180,E1 -12246.435,E2 -12246.435} C_VEL
LIN {X 0,Y 376.114,Z 393.636,A -85,B 0,C 180,E1 -12249.682,E2 -12249.682} C_VEL
LIN {X 0,Y 376.084,Z 393.636,A -85,B 0,C 180,E1 -12253.658,E2 -12253.658} C_VEL
LIN {X 0,Y 376.039,Z 393.645,A -85,B 0,C 180,E1 -12257.607,E2 -12257.607} C_VEL
LIN {X 0,Y 375.974,Z 393.654,A -85,B 0,C 180,E1 -12260.832,E2 -12260.832} C_VEL
LIN {X 0,Y 375.99,Z 393.652,A -85,B 0,C 180,E1 -12264.282,E2 -12264.282} C_VEL
LIN {X 0,Y 376.016,Z 393.645,A -85,B 0,C 180,E1 -12266.652,E2 -12266.652} C_VEL
LIN {X 0,Y 375.96,Z 393.658,A -85,B 0,C 180,E1 -12270.313,E2 -12270.313} C_VEL
LIN {X 0,Y 375.956,Z 393.66,A -85,B 0,C 180,E1 -12274.112,E2 -12274.112} C_VEL
LIN {X 0,Y 375.952,Z 393.659,A -85,B 0,C 180,E1 -12276.741,E2 -12276.741} C_VEL
LIN {X 0,Y 375.995,Z 393.652,A -85,B 0,C 180,E1 -12279.973,E2 -12279.973} C_VEL
LIN {X 0,Y 375.937,Z 393.66,A -85,B 0,C 180,E1 -12283.765,E2 -12283.765} C_VEL
LIN {X 0,Y 376.601,Z 397.144,A -85,B 0,C 180,E1 -12286.333,E2 -12286.333} C_VEL
LIN {X 0,Y 377.56,Z 402.469,A -85,B 0,C 180,E1 -12289.746,E2 -12289.746} C_VEL
LIN {X 0,Y 378.499,Z 407.978,A -85,B 0,C 180,E1 -12292.98,E2 -12292.98} C_VEL
LIN {X 0,Y 378.345,Z 411.455,A -85,B 0,C 180,E1 -12294.842,E2 -12294.842} C_VEL
LIN {X 0,Y 377.604,Z 417.681,A -85,B 0,C 180,E1 -12297.965,E2 -12297.965} C_VEL
LIN {X 0,Y 376.928,Z 424.395,A -85,B 0,C 180,E1 -12301.204,E2 -12301.204} C_VEL
LIN {X 0,Y 376.282,Z 431.614,A -85,B 0,C 180,E1 -12304.559,E2 -12304.559} C_VEL
LIN {X 0,Y 375.765,Z 439.341,A -85,B 0,C 180,E1 -12308.034,E2 -12308.034} C_VEL
LIN {X 0,Y 375.483,Z 445.184,A -85,B 0,C 180,E1 -12310.596,E2 -12310.596} C_VEL
LIN {X 0,Y 378.031,Z 459.921,A -85,B 0,C 180,E1 -12311.254,E2 -12311.254} C_VEL
LIN {X 0,Y 379.503,Z 472.507,A -85,B 0,C 180,E1 -12311.995,E2 -12311.995} C_VEL
LIN {X 0,Y 380.397,Z 480.691,A -85,B 0,C 180,E1 -12312.587,E2 -12312.587} C_VEL
LIN {X 0,Y 379.376,Z 492.982,A -85,B 0,C 180,E1 -12313.59,E2 -12313.59} C_VEL
LIN {X 0,Y 378.293,Z 504.489,A -85,B 0,C 180,E1 -12314.787,E2 -12314.787} C_VEL
LIN {X 0,Y 377.507,Z 513.793,A -85,B 0,C 180,E1 -12315.994,E2 -12315.994} C_VEL
LIN {X 0,Y 376.688,Z 522.309,A -85,B 0,C 180,E1 -12317.337,E2 -12317.337} C_VEL
LIN {X 0,Y 375.826,Z 530.646,A -85,B 0,C 180,E1 -12318.949,E2 -12318.949} C_VEL
LIN {X 0,Y 375.283,Z 537.387,A -85,B 0,C 180,E1 -12320.569,E2 -12320.569} C_VEL
LIN {X 0,Y 374.863,Z 543.565,A -85,B 0,C 180,E1 -12322.459,E2 -12322.459} C_VEL
LIN {X 0,Y 374.699,Z 546.892,A -85,B 0,C 180,E1 -12323.768,E2 -12323.768} C_VEL
LIN {X 0,Y 374.587,Z 550.578,A -85,B 0,C 180,E1 -12325.696,E2 -12325.696} C_VEL
LIN {X 0,Y 374.607,Z 553.023,A -85,B 0,C 180,E1 -12327.849,E2 -12327.849} C_VEL
LIN {X 0,Y 374.61,Z 553.65,A -85,B 0,C 180,E1 -12328.925,E2 -12328.925} C_VEL
LIN {X 0,Y 374.604,Z 553.872,A -85,B 0,C 180,E1 -12330,E2 -12330} C_VEL
LIN {X 0,Y 374.61,Z 553.655,A -85,B 0,C 180,E1 -12331.075,E2 -12331.075} C_VEL
LIN {X 0,Y 374.622,Z 553.046,A -85,B 0,C 180,E1 -12332.15,E2 -12332.15} C_VEL
LIN {X 0,Y 374.532,Z 552.036,A -85,B 0,C 180,E1 -12333.227,E2 -12333.227} C_VEL
LIN {X 0,Y 374.588,Z 550.618,A -85,B 0,C 180,E1 -12334.304,E2 -12334.304} C_VEL
LIN {X 0,Y 374.699,Z 546.934,A -85,B 0,C 180,E1 -12336.232,E2 -12336.232} C_VEL
LIN {X 0,Y 374.943,Z 542.001,A -85,B 0,C 180,E1 -12338.081,E2 -12338.081} C_VEL
LIN {X 0,Y 375.396,Z 536.406,A -85,B 0,C 180,E1 -12339.7,E2 -12339.7} C_VEL
LIN {X 0,Y 375.947,Z 529.419,A -85,B 0,C 180,E1 -12341.319,E2 -12341.319} C_VEL
LIN {X 0,Y 376.852,Z 520.677,A -85,B 0,C 180,E1 -12342.931,E2 -12342.931} C_VEL
LIN {X 0,Y 377.785,Z 511.061,A -85,B 0,C 180,E1 -12344.363,E2 -12344.363} C_VEL
LIN {X 0,Y 378.629,Z 500.701,A -85,B 0,C 180,E1 -12345.613,E2 -12345.613} C_VEL
LIN {X 0,Y 379.653,Z 489.567,A -85,B 0,C 180,E1 -12346.674,E2 -12346.674} C_VEL
LIN {X 0,Y 380.314,Z 480.129,A -85,B 0,C 180,E1 -12347.402,E2 -12347.402} C_VEL
LIN {X 0,Y 378.691,Z 466.421,A -85,B 0,C 180,E1 -12348.317,E2 -12348.317} C_VEL
LIN {X 0,Y 376.789,Z 453.649,A -85,B 0,C 180,E1 -12348.956,E2 -12348.956} C_VEL
LIN {X 0,Y 375.467,Z 446.009,A -85,B 0,C 180,E1 -12349.259,E2 -12349.259} C_VEL
LIN {X 0,Y 375.905,Z 438.591,A -85,B 0,C 180,E1 -12352.536,E2 -12352.536} C_VEL
LIN {X 0,Y 376.556,Z 430.051,A -85,B 0,C 180,E1 -12356.38,E2 -12356.38} C_VEL
LIN {X 0,Y 377.146,Z 423.137,A -85,B 0,C 180,E1 -12359.591,E2 -12359.591} C_VEL
LIN {X 0,Y 377.881,Z 415.652,A -85,B 0,C 180,E1 -12363.182,E2 -12363.182} C_VEL
LIN {X 0,Y 378.482,Z 410.381,A -85,B 0,C 180,E1 -12365.796,E2 -12365.796} C_VEL
LIN {X 0,Y 378.518,Z 407.978,A -85,B 0,C 180,E1 -12367.023,E2 -12367.023} C_VEL
LIN {X 0,Y 377.536,Z 402.156,A -85,B 0,C 180,E1 -12370.25,E2 -12370.25} C_VEL
LIN {X 0,Y 376.448,Z 396.314,A -85,B 0,C 180,E1 -12373.689,E2 -12373.689} C_VEL
LIN {X 0,Y 375.967,Z 393.655,A -85,B 0,C 180,E1 -12375.35,E2 -12375.35} C_VEL
LIN {X 0,Y 375.976,Z 393.655,A -85,B 0,C 180,E1 -12379.138,E2 -12379.138} C_VEL
LIN {X 0,Y 375.963,Z 393.655,A -85,B 0,C 180,E1 -12381.911,E2 -12381.911} C_VEL
LIN {X 0,Y 375.974,Z 393.652,A -85,B 0,C 180,E1 -12385.332,E2 -12385.332} C_VEL
LIN {X 0,Y 375.951,Z 393.654,A -85,B 0,C 180,E1 -12388.437,E2 -12388.437} C_VEL
LIN {X 0,Y 375.976,Z 393.65,A -85,B 0,C 180,E1 -12392.14,E2 -12392.14} C_VEL
LIN {X 0,Y 375.999,Z 393.65,A -85,B 0,C 180,E1 -12394.538,E2 -12394.538} C_VEL
LIN {X 0,Y 375.955,Z 393.652,A -85,B 0,C 180,E1 -12398.045,E2 -12398.045} C_VEL
LIN {X 0,Y 376.001,Z 393.647,A -85,B 0,C 180,E1 -12401.473,E2 -12401.473} C_VEL
LIN {X 0,Y 376.05,Z 393.646,A -85,B 0,C 180,E1 -12404.832,E2 -12404.832} C_VEL
LIN {X 0,Y 376.042,Z 393.642,A -85,B 0,C 180,E1 -12408.136,E2 -12408.136} C_VEL
LIN {X 0,Y 376.211,Z 393.621,A -85,B 0,C 180,E1 -12411.918,E2 -12411.918} C_VEL
LIN {X 0,Y 376.163,Z 393.631,A -85,B 0,C 180,E1 -12414.64,E2 -12414.64} C_VEL
LIN {X 0,Y 376.345,Z 393.604,A -85,B 0,C 180,E1 -12417.86,E2 -12417.86} C_VEL
LIN {X 0,Y 376.482,Z 393.587,A -85,B 0,C 180,E1 -12420,E2 -12420} C_VEL
LIN {X 0,Y 376.182,Z 393.625,A -85,B 0,C 180,E1 -12423.213,E2 -12423.213} C_VEL
LIN {X 0,Y 376.225,Z 393.621,A -85,B 0,C 180,E1 -12426.623,E2 -12426.623} C_VEL
LIN {X 0,Y 376.197,Z 393.627,A -85,B 0,C 180,E1 -12428.595,E2 -12428.595} C_VEL
LIN {X 0,Y 376.042,Z 393.642,A -85,B 0,C 180,E1 -12431.864,E2 -12431.864} C_VEL
LIN {X 0,Y 376.05,Z 393.641,A -85,B 0,C 180,E1 -12435.168,E2 -12435.168} C_VEL
LIN {X 0,Y 376.016,Z 393.649,A -85,B 0,C 180,E1 -12438.527,E2 -12438.527} C_VEL
LIN {X 0,Y 375.956,Z 393.654,A -85,B 0,C 180,E1 -12441.955,E2 -12441.955} C_VEL
LIN {X 0,Y 375.999,Z 393.646,A -85,B 0,C 180,E1 -12445.462,E2 -12445.462} C_VEL
LIN {X 0,Y 375.964,Z 393.651,A -85,B 0,C 180,E1 -12449.08,E2 -12449.08} C_VEL
LIN {X 0,Y 375.943,Z 393.655,A -85,B 0,C 180,E1 -12452.829,E2 -12452.829} C_VEL
LIN {X 0,Y 375.953,Z 393.652,A -85,B 0,C 180,E1 -12455.416,E2 -12455.416} C_VEL
LIN {X 0,Y 375.974,Z 393.655,A -85,B 0,C 180,E1 -12458.272,E2 -12458.272} C_VEL
LIN {X 0,Y 375.956,Z 393.653,A -85,B 0,C 180,E1 -12461.606,E2 -12461.606} C_VEL
LIN {X 0,Y 375.923,Z 393.656,A -85,B 0,C 180,E1 -12465.27,E2 -12465.27} C_VEL
LIN {X 0,Y 375.932,Z 393.659,A -85,B 0,C 180,E1 -12468.4,E2 -12468.4} C_VEL
LIN {X 0,Y 375.974,Z 393.652,A -85,B 0,C 180,E1 -12471.73,E2 -12471.73} C_VEL
LIN {X 0,Y 375.979,Z 393.65,A -85,B 0,C 180,E1 -12475.334,E2 -12475.334} C_VEL
LIN {X 0,Y 375.957,Z 393.654,A -85,B 0,C 180,E1 -12478.439,E2 -12478.439} C_VEL
LIN {X 0,Y 375.984,Z 393.653,A -85,B 0,C 180,E1 -12482.141,E2 -12482.141} C_VEL
LIN {X 0,Y 376.007,Z 393.647,A -85,B 0,C 180,E1 -12484.54,E2 -12484.54} C_VEL
LIN {X 0,Y 375.965,Z 393.656,A -85,B 0,C 180,E1 -12488.047,E2 -12488.047} C_VEL
LIN {X 0,Y 376.026,Z 393.645,A -85,B 0,C 180,E1 -12491.475,E2 -12491.475} C_VEL
LIN {X 0,Y 376.061,Z 393.639,A -85,B 0,C 180,E1 -12494.833,E2 -12494.833} C_VEL
LIN {X 0,Y 376.053,Z 393.643,A -85,B 0,C 180,E1 -12498.137,E2 -12498.137} C_VEL
LIN {X 0,Y 376.261,Z 393.619,A -85,B 0,C 180,E1 -12501.878,E2 -12501.878} C_VEL
LIN {X 0,Y 376.174,Z 393.625,A -85,B 0,C 180,E1 -12504.64,E2 -12504.64} C_VEL
LIN {X 0,Y 376.241,Z 393.622,A -85,B 0,C 180,E1 -12507.859,E2 -12507.859} C_VEL
LIN {X 0,Y 376.215,Z 393.621,A -85,B 0,C 180,E1 -12508.93,E2 -12508.93} C_VEL
LIN {X 0,Y 375.426,Z 393.724,A -85,B 0,C 180,E1 -12511.073,E2 -12511.073} C_VEL
LIN {X 0,Y 375.537,Z 396.42,A -85,B 0,C 180,E1 -12514.293,E2 -12514.293} C_VEL
LIN {X 0,Y 375.342,Z 399.507,A -85,B 0,C 180,E1 -12517.532,E2 -12517.532} C_VEL
LIN {X 0,Y 375.121,Z 402.726,A -85,B 0,C 180,E1 -12520.798,E2 -12520.798} C_VEL
LIN {X 0,Y 375.13,Z 404.973,A -85,B 0,C 180,E1 -12522.992,E2 -12522.992} C_VEL
LIN {X 0,Y 378.603,Z 418.111,A -85,B 0,C 180,E1 -12523.671,E2 -12523.671} C_VEL
LIN {X 0,Y 380.996,Z 428.972,A -85,B 0,C 180,E1 -12524.384,E2 -12524.384} C_VEL
LIN {X 0,Y 381.13,Z 432.455,A -85,B 0,C 180,E1 -12524.617,E2 -12524.617} C_VEL
LIN {X 0,Y 380.335,Z 444.016,A -85,B 0,C 180,E1 -12525.481,E2 -12525.481} C_VEL
LIN {X 0,Y 379.5,Z 455.148,A -85,B 0,C 180,E1 -12526.543,E2 -12526.543} C_VEL
LIN {X 0,Y 378.615,Z 464.879,A -85,B 0,C 180,E1 -12527.695,E2 -12527.695} C_VEL
LIN {X 0,Y 377.812,Z 473.854,A -85,B 0,C 180,E1 -12529.006,E2 -12529.006} C_VEL
LIN {X 0,Y 376.94,Z 482.041,A -85,B 0,C 180,E1 -12530.462,E2 -12530.462} C_VEL
LIN {X 0,Y 376.244,Z 488.808,A -85,B 0,C 180,E1 -12531.937,E2 -12531.937} C_VEL
LIN {X 0,Y 375.713,Z 494.841,A -85,B 0,C 180,E1 -12533.567,E2 -12533.567} C_VEL
LIN {X 0,Y 375.226,Z 500.397,A -85,B 0,C 180,E1 -12535.518,E2 -12535.518} C_VEL
LIN {X 0,Y 374.944,Z 504.136,A -85,B 0,C 180,E1 -12537.337,E2 -12537.337} C_VEL
LIN {X 0,Y 374.639,Z 506.689,A -85,B 0,C 180,E1 -12539.192,E2 -12539.192} C_VEL
LIN {X 0,Y 374.554,Z 507.74,A -85,B 0,C 180,E1 -12540.438,E2 -12540.438} C_VEL
LIN {X 0,Y 374.513,Z 507.978,A -85,B 0,C 180,E1 -12541.078,E2 -12541.078} C_VEL
LIN {X 0,Y 373.832,Z 508.302,A -85,B 0,C 180,E1 -12541.975,E2 -12541.975} C_VEL
LIN {X 0,Y 370.99,Z 508.232,A -85,B 0,C 180,E1 -12543.436,E2 -12543.436} C_VEL
LIN {X 0,Y 368.653,Z 507.704,A -85,B 0,C 180,E1 -12544.613,E2 -12544.613} C_VEL
LIN {X 0,Y 367.693,Z 506.779,A -85,B 0,C 180,E1 -12545.67,E2 -12545.67} C_VEL
LIN {X 0,Y 367.698,Z 506.515,A -85,B 0,C 180,E1 -12545.822,E2 -12545.822} C_VEL
LIN {X 0,Y 368.08,Z 503.794,A -85,B 0,C 180,E1 -12547.661,E2 -12547.661} C_VEL
LIN {X 0,Y 368.541,Z 499.32,A -85,B 0,C 180,E1 -12549.674,E2 -12549.674} C_VEL
LIN {X 0,Y 369.114,Z 494.072,A -85,B 0,C 180,E1 -12551.425,E2 -12551.425} C_VEL
LIN {X 0,Y 369.874,Z 487.369,A -85,B 0,C 180,E1 -12553.159,E2 -12553.159} C_VEL
LIN {X 0,Y 370.834,Z 478.856,A -85,B 0,C 180,E1 -12554.903,E2 -12554.903} C_VEL
LIN {X 0,Y 371.808,Z 470.346,A -85,B 0,C 180,E1 -12556.303,E2 -12556.303} C_VEL
LIN {X 0,Y 372.712,Z 461.141,A -85,B 0,C 180,E1 -12557.54,E2 -12557.54} C_VEL
LIN {X 0,Y 373.743,Z 449.629,A -85,B 0,C 180,E1 -12558.778,E2 -12558.778} C_VEL
LIN {X 0,Y 374.638,Z 438.84,A -85,B 0,C 180,E1 -12559.693,E2 -12559.693} C_VEL
LIN {X 0,Y 375.045,Z 432.961,A -85,B 0,C 180,E1 -12560.108,E2 -12560.108} C_VEL
LIN {X 0,Y 372.172,Z 420.424,A -85,B 0,C 180,E1 -12561.018,E2 -12561.018} C_VEL
LIN {X 0,Y 368.054,Z 406.723,A -85,B 0,C 180,E1 -12561.842,E2 -12561.842} C_VEL
LIN {X 0,Y 368.187,Z 403.726,A -85,B 0,C 180,E1 -12565.163,E2 -12565.163} C_VEL
LIN {X 0,Y 368.338,Z 401.466,A -85,B 0,C 180,E1 -12567.707,E2 -12567.707} C_VEL
LIN {X 0,Y 368.504,Z 398.153,A -85,B 0,C 180,E1 -12571.524,E2 -12571.524} C_VEL
LIN {X 0,Y 368.631,Z 396.063,A -85,B 0,C 180,E1 -12573.992,E2 -12573.992} C_VEL
LIN {X 0,Y 368.756,Z 394.557,A -85,B 0,C 180,E1 -12576.178,E2 -12576.178} C_VEL
LIN {X 0,Y 368.919,Z 394.535,A -85,B 0,C 180,E1 -12579.946,E2 -12579.946} C_VEL
LIN {X 0,Y 368.971,Z 394.527,A -85,B 0,C 180,E1 -12583.398,E2 -12583.398} C_VEL
LIN {X 0,Y 369.053,Z 394.516,A -85,B 0,C 180,E1 -12586.79,E2 -12586.79} C_VEL
LIN {X 0,Y 369.063,Z 394.514,A -85,B 0,C 180,E1 -12590.131,E2 -12590.131} C_VEL
LIN {X 0,Y 369.196,Z 394.498,A -85,B 0,C 180,E1 -12593.441,E2 -12593.441} C_VEL
LIN {X 0,Y 369.313,Z 394.481,A -85,B 0,C 180,E1 -12597.819,E2 -12597.819} C_VEL
LIN {X 0,Y 369.453,Z 394.462,A -85,B 0,C 180,E1 -12600,E2 -12600} C_VEL
LIN {X 0,Y 369.314,Z 394.48,A -85,B 0,C 180,E1 -12602.181,E2 -12602.181} C_VEL
LIN {X 0,Y 369.196,Z 394.499,A -85,B 0,C 180,E1 -12606.558,E2 -12606.558} C_VEL
LIN {X 0,Y 369.063,Z 394.514,A -85,B 0,C 180,E1 -12609.868,E2 -12609.868} C_VEL
LIN {X 0,Y 369.032,Z 394.515,A -85,B 0,C 180,E1 -12613.772,E2 -12613.772} C_VEL
LIN {X 0,Y 368.997,Z 394.522,A -85,B 0,C 180,E1 -12617.769,E2 -12617.769} C_VEL
LIN {X 0,Y 368.925,Z 394.532,A -85,B 0,C 180,E1 -12621.22,E2 -12621.22} C_VEL
LIN {X 0,Y 368.954,Z 394.528,A -85,B 0,C 180,E1 -12624.776,E2 -12624.776} C_VEL
LIN {X 0,Y 368.959,Z 394.527,A -85,B 0,C 180,E1 -12627.204,E2 -12627.204} C_VEL
LIN {X 0,Y 368.926,Z 394.531,A -85,B 0,C 180,E1 -12630.954,E2 -12630.954} C_VEL
LIN {X 0,Y 368.926,Z 394.533,A -85,B 0,C 180,E1 -12635.002,E2 -12635.002} C_VEL
LIN {X 0,Y 368.91,Z 394.535,A -85,B 0,C 180,E1 -12638.642,E2 -12638.642} C_VEL
LIN {X 0,Y 368.908,Z 394.533,A -85,B 0,C 180,E1 -12641.819,E2 -12641.819} C_VEL
LIN {X 0,Y 368.921,Z 394.733,A -85,B 0,C 180,E1 -12643.527,E2 -12643.527} C_VEL
LIN {X 0,Y 369.777,Z 399.373,A -85,B 0,C 180,E1 -12646.827,E2 -12646.827} C_VEL
LIN {X 0,Y 370.637,Z 404.048,A -85,B 0,C 180,E1 -12649.857,E2 -12649.857} C_VEL
LIN {X 0,Y 371.457,Z 408.833,A -85,B 0,C 180,E1 -12652.74,E2 -12652.74} C_VEL
LIN {X 0,Y 371.397,Z 411.953,A -85,B 0,C 180,E1 -12654.459,E2 -12654.459} C_VEL
LIN {X 0,Y 370.712,Z 417.391,A -85,B 0,C 180,E1 -12657.296,E2 -12657.296} C_VEL
LIN {X 0,Y 369.954,Z 424.707,A -85,B 0,C 180,E1 -12660.911,E2 -12660.911} C_VEL
LIN {X 0,Y 369.219,Z 432.558,A -85,B 0,C 180,E1 -12664.642,E2 -12664.642} C_VEL
LIN {X 0,Y 368.671,Z 440.27,A -85,B 0,C 180,E1 -12668.178,E2 -12668.178} C_VEL
LIN {X 0,Y 368.457,Z 444.982,A -85,B 0,C 180,E1 -12670.211,E2 -12670.211} C_VEL
LIN {X 0,Y 370.885,Z 458.596,A -85,B 0,C 180,E1 -12670.82,E2 -12670.82} C_VEL
LIN {X 0,Y 372.392,Z 470.548,A -85,B 0,C 180,E1 -12671.526,E2 -12671.526} C_VEL
LIN {X 0,Y 373.515,Z 481.9,A -85,B 0,C 180,E1 -12672.371,E2 -12672.371} C_VEL
LIN {X 0,Y 372.415,Z 494.126,A -85,B 0,C 180,E1 -12673.415,E2 -12673.415} C_VEL
LIN {X 0,Y 371.305,Z 505.284,A -85,B 0,C 180,E1 -12674.634,E2 -12674.634} C_VEL
LIN {X 0,Y 370.381,Z 515.249,A -85,B 0,C 180,E1 -12675.999,E2 -12675.999} C_VEL
LIN {X 0,Y 369.542,Z 523.443,A -85,B 0,C 180,E1 -12677.367,E2 -12677.367} C_VEL
LIN {X 0,Y 368.69,Z 531.506,A -85,B 0,C 180,E1 -12679.011,E2 -12679.011} C_VEL
LIN {X 0,Y 368.165,Z 537.985,A -85,B 0,C 180,E1 -12680.662,E2 -12680.662} C_VEL
LIN {X 0,Y 367.781,Z 543.147,A -85,B 0,C 180,E1 -12682.313,E2 -12682.313} C_VEL
LIN {X 0,Y 367.597,Z 546.857,A -85,B 0,C 180,E1 -12683.814,E2 -12683.814} C_VEL
LIN {X 0,Y 367.517,Z 550.155,A -85,B 0,C 180,E1 -12685.613,E2 -12685.613} C_VEL
LIN {X 0,Y 367.51,Z 552.597,A -85,B 0,C 180,E1 -12687.808,E2 -12687.808} C_VEL
LIN {X 0,Y 367.546,Z 553.225,A -85,B 0,C 180,E1 -12688.904,E2 -12688.904} C_VEL
LIN {X 0,Y 367.538,Z 553.442,A -85,B 0,C 180,E1 -12690,E2 -12690} C_VEL
LIN {X 0,Y 367.546,Z 553.223,A -85,B 0,C 180,E1 -12691.095,E2 -12691.095} C_VEL
LIN {X 0,Y 367.525,Z 552.61,A -85,B 0,C 180,E1 -12692.191,E2 -12692.191} C_VEL
LIN {X 0,Y 367.445,Z 551.598,A -85,B 0,C 180,E1 -12693.289,E2 -12693.289} C_VEL
LIN {X 0,Y 367.518,Z 550.175,A -85,B 0,C 180,E1 -12694.387,E2 -12694.387} C_VEL
LIN {X 0,Y 367.598,Z 546.858,A -85,B 0,C 180,E1 -12696.187,E2 -12696.187} C_VEL
LIN {X 0,Y 367.892,Z 541.542,A -85,B 0,C 180,E1 -12698.237,E2 -12698.237} C_VEL
LIN {X 0,Y 368.343,Z 535.938,A -85,B 0,C 180,E1 -12699.887,E2 -12699.887} C_VEL
LIN {X 0,Y 368.925,Z 528.939,A -85,B 0,C 180,E1 -12701.538,E2 -12701.538} C_VEL
LIN {X 0,Y 369.887,Z 520.185,A -85,B 0,C 180,E1 -12703.179,E2 -12703.179} C_VEL
LIN {X 0,Y 370.777,Z 511.418,A -85,B 0,C 180,E1 -12704.517,E2 -12704.517} C_VEL
LIN {X 0,Y 371.634,Z 501.373,A -85,B 0,C 180,E1 -12705.774,E2 -12705.774} C_VEL
LIN {X 0,Y 372.674,Z 490.568,A -85,B 0,C 180,E1 -12706.854,E2 -12706.854} C_VEL
LIN {X 0,Y 373.421,Z 481.037,A -85,B 0,C 180,E1 -12707.623,E2 -12707.623} C_VEL
LIN {X 0,Y 371.945,Z 468.056,A -85,B 0,C 180,E1 -12708.53,E2 -12708.53} C_VEL
LIN {X 0,Y 370.03,Z 454.695,A -85,B 0,C 180,E1 -12709.243,E2 -12709.243} C_VEL
LIN {X 0,Y 368.435,Z 445.65,A -85,B 0,C 180,E1 -12709.608,E2 -12709.608} C_VEL
LIN {X 0,Y 368.903,Z 438.189,A -85,B 0,C 180,E1 -12712.988,E2 -12712.988} C_VEL
LIN {X 0,Y 369.513,Z 430.306,A -85,B 0,C 180,E1 -12716.629,E2 -12716.629} C_VEL
LIN {X 0,Y 370.218,Z 422.789,A -85,B 0,C 180,E1 -12720.202,E2 -12720.202} C_VEL
LIN {X 0,Y 370.926,Z 416.045,A -85,B 0,C 180,E1 -12723.522,E2 -12723.522} C_VEL
LIN {X 0,Y 371.471,Z 411.317,A -85,B 0,C 180,E1 -12725.908,E2 -12725.908} C_VEL
LIN {X 0,Y 371.269,Z 407.491,A -85,B 0,C 180,E1 -12727.969,E2 -12727.969} C_VEL
LIN {X 0,Y 370.117,Z 401.087,A -85,B 0,C 180,E1 -12731.65,E2 -12731.65} C_VEL
LIN {X 0,Y 369.085,Z 395.307,A -85,B 0,C 180,E1 -12735.207,E2 -12735.207} C_VEL
LIN {X 0,Y 368.907,Z 394.535,A -85,B 0,C 180,E1 -12735.83,E2 -12735.83} C_VEL
LIN {X 0,Y 368.948,Z 394.529,A -85,B 0,C 180,E1 -12739.635,E2 -12739.635} C_VEL
LIN {X 0,Y 368.898,Z 394.536,A -85,B 0,C 180,E1 -12743.143,E2 -12743.143} C_VEL
LIN {X 0,Y 368.89,Z 394.534,A -85,B 0,C 180,E1 -12746.461,E2 -12746.461} C_VEL
LIN {X 0,Y 368.923,Z 394.533,A -85,B 0,C 180,E1 -12749.046,E2 -12749.046} C_VEL
LIN {X 0,Y 368.956,Z 394.529,A -85,B 0,C 180,E1 -12752.796,E2 -12752.796} C_VEL
LIN {X 0,Y 368.938,Z 394.526,A -85,B 0,C 180,E1 -12756.113,E2 -12756.113} C_VEL
LIN {X 0,Y 368.928,Z 394.527,A -85,B 0,C 180,E1 -12759.947,E2 -12759.947} C_VEL
LIN {X 0,Y 368.967,Z 394.523,A -85,B 0,C 180,E1 -12763.398,E2 -12763.398} C_VEL
LIN {X 0,Y 369.049,Z 394.517,A -85,B 0,C 180,E1 -12766.79,E2 -12766.79} C_VEL
LIN {X 0,Y 369.059,Z 394.512,A -85,B 0,C 180,E1 -12770.132,E2 -12770.132} C_VEL
LIN {X 0,Y 369.192,Z 394.495,A -85,B 0,C 180,E1 -12773.442,E2 -12773.442} C_VEL
LIN {X 0,Y 369.31,Z 394.48,A -85,B 0,C 180,E1 -12777.819,E2 -12777.819} C_VEL
LIN {X 0,Y 369.452,Z 394.463,A -85,B 0,C 180,E1 -12780,E2 -12780} C_VEL
LIN {X 0,Y 369.311,Z 394.482,A -85,B 0,C 180,E1 -12782.181,E2 -12782.181} C_VEL
LIN {X 0,Y 369.196,Z 394.498,A -85,B 0,C 180,E1 -12786.61,E2 -12786.61} C_VEL
LIN {X 0,Y 369.13,Z 394.506,A -85,B 0,C 180,E1 -12788.761,E2 -12788.761} C_VEL
LIN {X 0,Y 368.998,Z 394.521,A -85,B 0,C 180,E1 -12792.094,E2 -12792.094} C_VEL
LIN {X 0,Y 368.99,Z 394.519,A -85,B 0,C 180,E1 -12795.465,E2 -12795.465} C_VEL
LIN {X 0,Y 368.975,Z 394.523,A -85,B 0,C 180,E1 -12798.893,E2 -12798.893} C_VEL
LIN {X 0,Y 368.925,Z 394.533,A -85,B 0,C 180,E1 -12802.396,E2 -12802.396} C_VEL
LIN {X 0,Y 368.993,Z 394.521,A -85,B 0,C 180,E1 -12805.981,E2 -12805.981} C_VEL
LIN {X 0,Y 368.955,Z 394.526,A -85,B 0,C 180,E1 -12808.812,E2 -12808.812} C_VEL
LIN {X 0,Y 368.892,Z 394.537,A -85,B 0,C 180,E1 -12812.239,E2 -12812.239} C_VEL
LIN {X 0,Y 368.924,Z 394.528,A -85,B 0,C 180,E1 -12815.002,E2 -12815.002} C_VEL
LIN {X 0,Y 368.909,Z 394.532,A -85,B 0,C 180,E1 -12818.642,E2 -12818.642} C_VEL
LIN {X 0,Y 368.906,Z 394.533,A -85,B 0,C 180,E1 -12821.82,E2 -12821.82} C_VEL
LIN {X 0,Y 368.876,Z 394.533,A -85,B 0,C 180,E1 -12825.177,E2 -12825.177} C_VEL
LIN {X 0,Y 368.881,Z 394.538,A -85,B 0,C 180,E1 -12828.179,E2 -12828.179} C_VEL
LIN {X 0,Y 368.908,Z 394.53,A -85,B 0,C 180,E1 -12831.36,E2 -12831.36} C_VEL
LIN {X 0,Y 368.936,Z 394.526,A -85,B 0,C 180,E1 -12835.148,E2 -12835.148} C_VEL
LIN {X 0,Y 368.929,Z 394.527,A -85,B 0,C 180,E1 -12839.047,E2 -12839.047} C_VEL
LIN {X 0,Y 368.964,Z 394.523,A -85,B 0,C 180,E1 -12842.797,E2 -12842.797} C_VEL
LIN {X 0,Y 368.947,Z 394.53,A -85,B 0,C 180,E1 -12846.114,E2 -12846.114} C_VEL
LIN {X 0,Y 368.939,Z 394.531,A -85,B 0,C 180,E1 -12849.948,E2 -12849.948} C_VEL
LIN {X 0,Y 368.978,Z 394.523,A -85,B 0,C 180,E1 -12853.399,E2 -12853.399} C_VEL
LIN {X 0,Y 369.06,Z 394.511,A -85,B 0,C 180,E1 -12856.791,E2 -12856.791} C_VEL
LIN {X 0,Y 369.07,Z 394.512,A -85,B 0,C 180,E1 -12860.132,E2 -12860.132} C_VEL
LIN {X 0,Y 369.192,Z 394.496,A -85,B 0,C 180,E1 -12862.343,E2 -12862.343} C_VEL
LIN {X 0,Y 369.147,Z 394.5,A -85,B 0,C 180,E1 -12864.538,E2 -12864.538} C_VEL
LIN {X 0,Y 369.184,Z 394.501,A -85,B 0,C 180,E1 -12867.818,E2 -12867.818} C_VEL
LIN {X 0,Y 369.185,Z 394.496,A -85,B 0,C 180,E1 -12868.91,E2 -12868.91} C_VEL
LIN {X 0,Y 368.371,Z 394.603,A -85,B 0,C 180,E1 -12871.093,E2 -12871.093} C_VEL
LIN {X 0,Y 368.498,Z 397.335,A -85,B 0,C 180,E1 -12874.375,E2 -12874.375} C_VEL
LIN {X 0,Y 368.281,Z 400.41,A -85,B 0,C 180,E1 -12877.677,E2 -12877.677} C_VEL
LIN {X 0,Y 368.045,Z 403.665,A -85,B 0,C 180,E1 -12881.009,E2 -12881.009} C_VEL
LIN {X 0,Y 368.079,Z 405.309,A -85,B 0,C 180,E1 -12882.635,E2 -12882.635} C_VEL
LIN {X 0,Y 371.518,Z 418.442,A -85,B 0,C 180,E1 -12883.327,E2 -12883.327} C_VEL
LIN {X 0,Y 374.37,Z 431.236,A -85,B 0,C 180,E1 -12884.198,E2 -12884.198} C_VEL
LIN {X 0,Y 373.678,Z 442.288,A -85,B 0,C 180,E1 -12885.006,E2 -12885.006} C_VEL
LIN {X 0,Y 372.732,Z 454.463,A -85,B 0,C 180,E1 -12886.154,E2 -12886.154} C_VEL
LIN {X 0,Y 371.843,Z 464.328,A -85,B 0,C 180,E1 -12887.318,E2 -12887.318} C_VEL
LIN {X 0,Y 370.876,Z 474.367,A -85,B 0,C 180,E1 -12888.793,E2 -12888.793} C_VEL
LIN {X 0,Y 369.983,Z 482.575,A -85,B 0,C 180,E1 -12890.283,E2 -12890.283} C_VEL
LIN {X 0,Y 369.168,Z 490.536,A -85,B 0,C 180,E1 -12892.085,E2 -12892.085} C_VEL
LIN {X 0,Y 368.604,Z 496.352,A -85,B 0,C 180,E1 -12893.766,E2 -12893.766} C_VEL
LIN {X 0,Y 368.162,Z 500.885,A -85,B 0,C 180,E1 -12895.436,E2 -12895.436} C_VEL
LIN {X 0,Y 367.885,Z 504.608,A -85,B 0,C 180,E1 -12897.289,E2 -12897.289} C_VEL
LIN {X 0,Y 367.633,Z 506.46,A -85,B 0,C 180,E1 -12898.549,E2 -12898.549} C_VEL
LIN {X 0,Y 367.477,Z 508.261,A -85,B 0,C 180,E1 -12900.612,E2 -12900.612} C_VEL
LIN {X 0,Y 367.452,Z 508.66,A -85,B 0,C 180,E1 -12902.694,E2 -12902.694} C_VEL
LIN {X 0,Y 367.566,Z 507.722,A -85,B 0,C 180,E1 -12904.696,E2 -12904.696} C_VEL
LIN {X 0,Y 367.698,Z 506.515,A -85,B 0,C 180,E1 -12905.822,E2 -12905.822} C_VEL
LIN {X 0,Y 367.206,Z 505.43,A -85,B 0,C 180,E1 -12906.723,E2 -12906.723} C_VEL
LIN {X 0,Y 364.68,Z 503.164,A -85,B 0,C 180,E1 -12908.183,E2 -12908.183} C_VEL
LIN {X 0,Y 362.56,Z 500.876,A -85,B 0,C 180,E1 -12909.34,E2 -12909.34} C_VEL
LIN {X 0,Y 361.754,Z 498.779,A -85,B 0,C 180,E1 -12910.21,E2 -12910.21} C_VEL
LIN {X 0,Y 361.747,Z 497.979,A -85,B 0,C 180,E1 -12910.498,E2 -12910.498} C_VEL
LIN {X 0,Y 362.404,Z 492.377,A -85,B 0,C 180,E1 -12912.234,E2 -12912.234} C_VEL
LIN {X 0,Y 363.155,Z 486.149,A -85,B 0,C 180,E1 -12913.776,E2 -12913.776} C_VEL
LIN {X 0,Y 363.981,Z 479.014,A -85,B 0,C 180,E1 -12915.224,E2 -12915.224} C_VEL
LIN {X 0,Y 365.04,Z 469.902,A -85,B 0,C 180,E1 -12916.728,E2 -12916.728} C_VEL
LIN {X 0,Y 366.046,Z 460.445,A -85,B 0,C 180,E1 -12917.992,E2 -12917.992} C_VEL
LIN {X 0,Y 367.023,Z 450.037,A -85,B 0,C 180,E1 -12919.121,E2 -12919.121} C_VEL
LIN {X 0,Y 368.033,Z 438.194,A -85,B 0,C 180,E1 -12920.134,E2 -12920.134} C_VEL
LIN {X 0,Y 368.191,Z 433.634,A -85,B 0,C 180,E1 -12920.466,E2 -12920.466} C_VEL
LIN {X 0,Y 365.397,Z 421.564,A -85,B 0,C 180,E1 -12921.377,E2 -12921.377} C_VEL
LIN {X 0,Y 361.519,Z 409.275,A -85,B 0,C 180,E1 -12922.151,E2 -12922.151} C_VEL
LIN {X 0,Y 361.014,Z 407.198,A -85,B 0,C 180,E1 -12922.265,E2 -12922.265} C_VEL
LIN {X 0,Y 361.163,Z 404.205,A -85,B 0,C 180,E1 -12925.645,E2 -12925.645} C_VEL
LIN {X 0,Y 361.338,Z 401.42,A -85,B 0,C 180,E1 -12928.846,E2 -12928.846} C_VEL
LIN {X 0,Y 361.481,Z 398.588,A -85,B 0,C 180,E1 -12932.185,E2 -12932.185} C_VEL
LIN {X 0,Y 361.681,Z 395.486,A -85,B 0,C 180,E1 -12935.961,E2 -12935.961} C_VEL
LIN {X 0,Y 361.874,Z 395.414,A -85,B 0,C 180,E1 -12939.538,E2 -12939.538} C_VEL
LIN {X 0,Y 361.929,Z 395.403,A -85,B 0,C 180,E1 -12943.066,E2 -12943.066} C_VEL
LIN {X 0,Y 361.994,Z 395.396,A -85,B 0,C 180,E1 -12946.527,E2 -12946.527} C_VEL
LIN {X 0,Y 362.027,Z 395.39,A -85,B 0,C 180,E1 -12949.938,E2 -12949.938} C_VEL
LIN {X 0,Y 362.158,Z 395.375,A -85,B 0,C 180,E1 -12953.313,E2 -12953.313} C_VEL
LIN {X 0,Y 362.277,Z 395.357,A -85,B 0,C 180,E1 -12957.776,E2 -12957.776} C_VEL
LIN {X 0,Y 362.422,Z 395.338,A -85,B 0,C 180,E1 -12960,E2 -12960} C_VEL
LIN {X 0,Y 362.277,Z 395.357,A -85,B 0,C 180,E1 -12962.223,E2 -12962.223} C_VEL
LIN {X 0,Y 362.157,Z 395.375,A -85,B 0,C 180,E1 -12966.686,E2 -12966.686} C_VEL
LIN {X 0,Y 362.027,Z 395.388,A -85,B 0,C 180,E1 -12970.062,E2 -12970.062} C_VEL
LIN {X 0,Y 361.993,Z 395.392,A -85,B 0,C 180,E1 -12973.899,E2 -12973.899} C_VEL
LIN {X 0,Y 361.963,Z 395.398,A -85,B 0,C 180,E1 -12977.939,E2 -12977.939} C_VEL
LIN {X 0,Y 361.888,Z 395.408,A -85,B 0,C 180,E1 -12981.653,E2 -12981.653} C_VEL
LIN {X 0,Y 361.924,Z 395.404,A -85,B 0,C 180,E1 -12985.29,E2 -12985.29} C_VEL
LIN {X 0,Y 361.904,Z 395.407,A -85,B 0,C 180,E1 -12987.779,E2 -12987.779} C_VEL
LIN {X 0,Y 361.834,Z 395.416,A -85,B 0,C 180,E1 -12991.63,E2 -12991.63} C_VEL
LIN {X 0,Y 361.871,Z 395.412,A -85,B 0,C 180,E1 -12995.345,E2 -12995.345} C_VEL
LIN {X 0,Y 361.872,Z 395.412,A -85,B 0,C 180,E1 -12999.028,E2 -12999.028} C_VEL
LIN {X 0,Y 361.854,Z 395.414,A -85,B 0,C 180,E1 -13002.436,E2 -13002.436} C_VEL
LIN {X 0,Y 361.885,Z 395.617,A -85,B 0,C 180,E1 -13003.012,E2 -13003.012} C_VEL
LIN {X 0,Y 362.776,Z 400.486,A -85,B 0,C 180,E1 -13006.577,E2 -13006.577} C_VEL
LIN {X 0,Y 363.634,Z 405.154,A -85,B 0,C 180,E1 -13009.68,E2 -13009.68} C_VEL
LIN {X 0,Y 364.346,Z 409.319,A -85,B 0,C 180,E1 -13012.267,E2 -13012.267} C_VEL
LIN {X 0,Y 364.477,Z 412.484,A -85,B 0,C 180,E1 -13014.083,E2 -13014.083} C_VEL
LIN {X 0,Y 363.703,Z 418.396,A -85,B 0,C 180,E1 -13017.245,E2 -13017.245} C_VEL
LIN {X 0,Y 362.953,Z 425.045,A -85,B 0,C 180,E1 -13020.616,E2 -13020.616} C_VEL
LIN {X 0,Y 362.272,Z 432.227,A -85,B 0,C 180,E1 -13024.12,E2 -13024.12} C_VEL
LIN {X 0,Y 361.598,Z 441.175,A -85,B 0,C 180,E1 -13028.329,E2 -13028.329} C_VEL
LIN {X 0,Y 361.417,Z 444.296,A -85,B 0,C 180,E1 -13029.772,E2 -13029.772} C_VEL
LIN {X 0,Y 363.944,Z 458.078,A -85,B 0,C 180,E1 -13030.411,E2 -13030.411} C_VEL
LIN {X 0,Y 365.487,Z 470.413,A -85,B 0,C 180,E1 -13031.164,E2 -13031.164} C_VEL
LIN {X 0,Y 366.661,Z 483.009,A -85,B 0,C 180,E1 -13032.141,E2 -13032.141} C_VEL
LIN {X 0,Y 365.599,Z 493.842,A -85,B 0,C 180,E1 -13033.097,E2 -13033.097} C_VEL
LIN {X 0,Y 364.444,Z 504.959,A -85,B 0,C 180,E1 -13034.337,E2 -13034.337} C_VEL
LIN {X 0,Y 363.474,Z 514.904,A -85,B 0,C 180,E1 -13035.728,E2 -13035.728} C_VEL
LIN {X 0,Y 362.406,Z 524.572,A -85,B 0,C 180,E1 -13037.399,E2 -13037.399} C_VEL
LIN {X 0,Y 361.586,Z 532.287,A -85,B 0,C 180,E1 -13039.076,E2 -13039.076} C_VEL
LIN {X 0,Y 360.97,Z 539.441,A -85,B 0,C 180,E1 -13041.039,E2 -13041.039} C_VEL
LIN {X 0,Y 360.622,Z 544.206,A -85,B 0,C 180,E1 -13042.722,E2 -13042.722} C_VEL
LIN {X 0,Y 360.466,Z 547.857,A -85,B 0,C 180,E1 -13044.405,E2 -13044.405} C_VEL
LIN {X 0,Y 360.447,Z 549.739,A -85,B 0,C 180,E1 -13045.527,E2 -13045.527} C_VEL
LIN {X 0,Y 360.414,Z 552.173,A -85,B 0,C 180,E1 -13047.765,E2 -13047.765} C_VEL
LIN {X 0,Y 360.482,Z 552.8,A -85,B 0,C 180,E1 -13048.883,E2 -13048.883} C_VEL
LIN {X 0,Y 360.473,Z 553.012,A -85,B 0,C 180,E1 -13050,E2 -13050} C_VEL
LIN {X 0,Y 360.483,Z 552.79,A -85,B 0,C 180,E1 -13051.117,E2 -13051.117} C_VEL
LIN {X 0,Y 360.428,Z 552.172,A -85,B 0,C 180,E1 -13052.235,E2 -13052.235} C_VEL
LIN {X 0,Y 360.363,Z 551.157,A -85,B 0,C 180,E1 -13053.354,E2 -13053.354} C_VEL
LIN {X 0,Y 360.449,Z 549.728,A -85,B 0,C 180,E1 -13054.473,E2 -13054.473} C_VEL
LIN {X 0,Y 360.526,Z 546.679,A -85,B 0,C 180,E1 -13056.184,E2 -13056.184} C_VEL
LIN {X 0,Y 360.718,Z 542.694,A -85,B 0,C 180,E1 -13057.838,E2 -13057.838} C_VEL
LIN {X 0,Y 361.224,Z 536.469,A -85,B 0,C 180,E1 -13059.801,E2 -13059.801} C_VEL
LIN {X 0,Y 361.82,Z 529.685,A -85,B 0,C 180,E1 -13061.484,E2 -13061.484} C_VEL
LIN {X 0,Y 362.781,Z 521.281,A -85,B 0,C 180,E1 -13063.157,E2 -13063.157} C_VEL
LIN {X 0,Y 363.818,Z 511.317,A -85,B 0,C 180,E1 -13064.734,E2 -13064.734} C_VEL
LIN {X 0,Y 364.739,Z 500.784,A -85,B 0,C 180,E1 -13066.08,E2 -13066.08} C_VEL
LIN {X 0,Y 365.861,Z 489.926,A -85,B 0,C 180,E1 -13067.178,E2 -13067.178} C_VEL
LIN {X 0,Y 366.494,Z 481.601,A -85,B 0,C 180,E1 -13067.867,E2 -13067.867} C_VEL
LIN {X 0,Y 365.151,Z 469.447,A -85,B 0,C 180,E1 -13068.766,E2 -13068.766} C_VEL
LIN {X 0,Y 363.244,Z 455.93,A -85,B 0,C 180,E1 -13069.529,E2 -13069.529} C_VEL
LIN {X 0,Y 361.42,Z 445.209,A -85,B 0,C 180,E1 -13070.005,E2 -13070.005} C_VEL
LIN {X 0,Y 361.889,Z 437.771,A -85,B 0,C 180,E1 -13073.46,E2 -13073.46} C_VEL
LIN {X 0,Y 362.487,Z 430.521,A -85,B 0,C 180,E1 -13076.892,E2 -13076.892} C_VEL
LIN {X 0,Y 363.188,Z 423.697,A -85,B 0,C 180,E1 -13080.206,E2 -13080.206} C_VEL
LIN {X 0,Y 363.849,Z 417.495,A -85,B 0,C 180,E1 -13083.313,E2 -13083.313} C_VEL
LIN {X 0,Y 364.447,Z 412.469,A -85,B 0,C 180,E1 -13085.911,E2 -13085.911} C_VEL
LIN {X 0,Y 364.23,Z 408.417,A -85,B 0,C 180,E1 -13088.129,E2 -13088.129} C_VEL
LIN {X 0,Y 363.1,Z 402.097,A -85,B 0,C 180,E1 -13091.859,E2 -13091.859} C_VEL
LIN {X 0,Y 362.007,Z 396.068,A -85,B 0,C 180,E1 -13095.661,E2 -13095.661} C_VEL
LIN {X 0,Y 361.87,Z 395.411,A -85,B 0,C 180,E1 -13096.239,E2 -13096.239} C_VEL
LIN {X 0,Y 361.876,Z 395.409,A -85,B 0,C 180,E1 -13100.141,E2 -13100.141} C_VEL
LIN {X 0,Y 361.864,Z 395.413,A -85,B 0,C 180,E1 -13102.982,E2 -13102.982} C_VEL
LIN {X 0,Y 361.852,Z 395.412,A -85,B 0,C 180,E1 -13106.63,E2 -13106.63} C_VEL
LIN {X 0,Y 361.866,Z 395.407,A -85,B 0,C 180,E1 -13109.671,E2 -13109.671} C_VEL
LIN {X 0,Y 361.947,Z 395.398,A -85,B 0,C 180,E1 -13113.474,E2 -13113.474} C_VEL
LIN {X 0,Y 361.882,Z 395.408,A -85,B 0,C 180,E1 -13117.144,E2 -13117.144} C_VEL
LIN {X 0,Y 361.899,Z 395.408,A -85,B 0,C 180,E1 -13120.723,E2 -13120.723} C_VEL
LIN {X 0,Y 361.925,Z 395.403,A -85,B 0,C 180,E1 -13123.066,E2 -13123.066} C_VEL
LIN {X 0,Y 361.991,Z 395.395,A -85,B 0,C 180,E1 -13126.528,E2 -13126.528} C_VEL
LIN {X 0,Y 362.023,Z 395.387,A -85,B 0,C 180,E1 -13129.938,E2 -13129.938} C_VEL
LIN {X 0,Y 362.154,Z 395.372,A -85,B 0,C 180,E1 -13133.314,E2 -13133.314} C_VEL
LIN {X 0,Y 362.274,Z 395.356,A -85,B 0,C 180,E1 -13137.777,E2 -13137.777} C_VEL
LIN {X 0,Y 362.421,Z 395.339,A -85,B 0,C 180,E1 -13140,E2 -13140} C_VEL
LIN {X 0,Y 362.275,Z 395.359,A -85,B 0,C 180,E1 -13142.224,E2 -13142.224} C_VEL
LIN {X 0,Y 362.163,Z 395.375,A -85,B 0,C 180,E1 -13146.686,E2 -13146.686} C_VEL
LIN {X 0,Y 362.066,Z 395.384,A -85,B 0,C 180,E1 -13148.934,E2 -13148.934} C_VEL
LIN {X 0,Y 361.953,Z 395.401,A -85,B 0,C 180,E1 -13152.333,E2 -13152.333} C_VEL
LIN {X 0,Y 361.954,Z 395.4,A -85,B 0,C 180,E1 -13154.621,E2 -13154.621} C_VEL
LIN {X 0,Y 361.952,Z 395.399,A -85,B 0,C 180,E1 -13158.1,E2 -13158.1} C_VEL
LIN {X 0,Y 361.885,Z 395.405,A -85,B 0,C 180,E1 -13161.654,E2 -13161.654} C_VEL
LIN {X 0,Y 361.922,Z 395.4,A -85,B 0,C 180,E1 -13165.291,E2 -13165.291} C_VEL
LIN {X 0,Y 361.912,Z 395.402,A -85,B 0,C 180,E1 -13167.779,E2 -13167.779} C_VEL
LIN {X 0,Y 361.841,Z 395.41,A -85,B 0,C 180,E1 -13171.286,E2 -13171.286} C_VEL
LIN {X 0,Y 361.849,Z 395.414,A -85,B 0,C 180,E1 -13174.281,E2 -13174.281} C_VEL
LIN {X 0,Y 361.861,Z 395.407,A -85,B 0,C 180,E1 -13177.224,E2 -13177.224} C_VEL
LIN {X 0,Y 361.868,Z 395.408,A -85,B 0,C 180,E1 -13180.763,E2 -13180.763} C_VEL
LIN {X 0,Y 361.819,Z 395.417,A -85,B 0,C 180,E1 -13184.369,E2 -13184.369} C_VEL
LIN {X 0,Y 361.833,Z 395.412,A -85,B 0,C 180,E1 -13187.569,E2 -13187.569} C_VEL
LIN {X 0,Y 361.869,Z 395.406,A -85,B 0,C 180,E1 -13190.974,E2 -13190.974} C_VEL
LIN {X 0,Y 361.873,Z 395.407,A -85,B 0,C 180,E1 -13194.656,E2 -13194.656} C_VEL
LIN {X 0,Y 361.837,Z 395.413,A -85,B 0,C 180,E1 -13198.372,E2 -13198.372} C_VEL
LIN {X 0,Y 361.909,Z 395.405,A -85,B 0,C 180,E1 -13202.222,E2 -13202.222} C_VEL
LIN {X 0,Y 361.929,Z 395.399,A -85,B 0,C 180,E1 -13204.711,E2 -13204.711} C_VEL
LIN {X 0,Y 361.893,Z 395.406,A -85,B 0,C 180,E1 -13208.348,E2 -13208.348} C_VEL
LIN {X 0,Y 361.969,Z 395.398,A -85,B 0,C 180,E1 -13212.062,E2 -13212.062} C_VEL
LIN {X 0,Y 362,Z 395.394,A -85,B 0,C 180,E1 -13216.102,E2 -13216.102} C_VEL
LIN {X 0,Y 362.034,Z 395.391,A -85,B 0,C 180,E1 -13219.939,E2 -13219.939} C_VEL
LIN {X 0,Y 362.155,Z 395.373,A -85,B 0,C 180,E1 -13222.193,E2 -13222.193} C_VEL
LIN {X 0,Y 362.121,Z 395.376,A -85,B 0,C 180,E1 -13224.432,E2 -13224.432} C_VEL
LIN {X 0,Y 362.154,Z 395.372,A -85,B 0,C 180,E1 -13228.888,E2 -13228.888} C_VEL
LIN {X 0,Y 361.316,Z 395.482,A -85,B 0,C 180,E1 -13231.115,E2 -13231.115} C_VEL
LIN {X 0,Y 361.439,Z 398.246,A -85,B 0,C 180,E1 -13234.461,E2 -13234.461} C_VEL
LIN {X 0,Y 361.232,Z 401.408,A -85,B 0,C 180,E1 -13237.828,E2 -13237.828} C_VEL
LIN {X 0,Y 361.006,Z 405.614,A -85,B 0,C 180,E1 -13242.258,E2 -13242.258} C_VEL
LIN {X 0,Y 364.677,Z 419.393,A -85,B 0,C 180,E1 -13243.014,E2 -13243.014} C_VEL
LIN {X 0,Y 367.401,Z 431.677,A -85,B 0,C 180,E1 -13243.875,E2 -13243.875} C_VEL
LIN {X 0,Y 367.488,Z 434.475,A -85,B 0,C 180,E1 -13244.081,E2 -13244.081} C_VEL
LIN {X 0,Y 366.634,Z 446.037,A -85,B 0,C 180,E1 -13244.998,E2 -13244.998} C_VEL
LIN {X 0,Y 365.724,Z 456.839,A -85,B 0,C 180,E1 -13246.087,E2 -13246.087} C_VEL
LIN {X 0,Y 364.718,Z 467.061,A -85,B 0,C 180,E1 -13247.378,E2 -13247.378} C_VEL
LIN {X 0,Y 363.702,Z 476.853,A -85,B 0,C 180,E1 -13248.912,E2 -13248.912} C_VEL
LIN {X 0,Y 362.829,Z 484.587,A -85,B 0,C 180,E1 -13250.405,E2 -13250.405} C_VEL
LIN {X 0,Y 362.165,Z 491.038,A -85,B 0,C 180,E1 -13251.935,E2 -13251.935} C_VEL
LIN {X 0,Y 361.623,Z 496.132,A -85,B 0,C 180,E1 -13253.413,E2 -13253.413} C_VEL
LIN {X 0,Y 361.098,Z 501.365,A -85,B 0,C 180,E1 -13255.352,E2 -13255.352} C_VEL
LIN {X 0,Y 360.834,Z 505.07,A -85,B 0,C 180,E1 -13257.239,E2 -13257.239} C_VEL
LIN {X 0,Y 360.475,Z 507.606,A -85,B 0,C 180,E1 -13259.17,E2 -13259.17} C_VEL
LIN {X 0,Y 360.376,Z 508.829,A -85,B 0,C 180,E1 -13260.897,E2 -13260.897} C_VEL
LIN {X 0,Y 360.377,Z 509.046,A -85,B 0,C 180,E1 -13263.096,E2 -13263.096} C_VEL
LIN {X 0,Y 360.543,Z 507.918,A -85,B 0,C 180,E1 -13265.045,E2 -13265.045} C_VEL
LIN {X 0,Y 360.904,Z 505.347,A -85,B 0,C 180,E1 -13267.133,E2 -13267.133} C_VEL
LIN {X 0,Y 361.284,Z 501.988,A -85,B 0,C 180,E1 -13268.911,E2 -13268.911} C_VEL
LIN {X 0,Y 361.747,Z 497.979,A -85,B 0,C 180,E1 -13270.498,E2 -13270.498} C_VEL
LIN {X 0,Y 361.334,Z 495.545,A -85,B 0,C 180,E1 -13271.351,E2 -13271.351} C_VEL
LIN {X 0,Y 359.004,Z 491.308,A -85,B 0,C 180,E1 -13272.734,E2 -13272.734} C_VEL
LIN {X 0,Y 356.84,Z 486.393,A -85,B 0,C 180,E1 -13274.068,E2 -13274.068} C_VEL
LIN {X 0,Y 356.677,Z 482.905,A -85,B 0,C 180,E1 -13274.832,E2 -13274.832} C_VEL
LIN {X 0,Y 357.827,Z 473.85,A -85,B 0,C 180,E1 -13276.486,E2 -13276.486} C_VEL
LIN {X 0,Y 358.911,Z 464.451,A -85,B 0,C 180,E1 -13277.871,E2 -13277.871} C_VEL
LIN {X 0,Y 360.028,Z 453.324,A -85,B 0,C 180,E1 -13279.192,E2 -13279.192} C_VEL
LIN {X 0,Y 361.072,Z 442.048,A -85,B 0,C 180,E1 -13280.234,E2 -13280.234} C_VEL
LIN {X 0,Y 361.576,Z 435.744,A -85,B 0,C 180,E1 -13280.714,E2 -13280.714} C_VEL
LIN {X 0,Y 359.186,Z 424.807,A -85,B 0,C 180,E1 -13281.593,E2 -13281.593} C_VEL
LIN {X 0,Y 355.59,Z 412.751,A -85,B 0,C 180,E1 -13282.421,E2 -13282.421} C_VEL
LIN {X 0,Y 353.982,Z 407.668,A -85,B 0,C 180,E1 -13282.723,E2 -13282.723} C_VEL
LIN {X 0,Y 354.174,Z 404.418,A -85,B 0,C 180,E1 -13286.45,E2 -13286.45} C_VEL
LIN {X 0,Y 354.304,Z 402.285,A -85,B 0,C 180,E1 -13288.953,E2 -13288.953} C_VEL
LIN {X 0,Y 354.455,Z 400.095,A -85,B 0,C 180,E1 -13291.584,E2 -13291.584} C_VEL
LIN {X 0,Y 354.654,Z 396.729,A -85,B 0,C 180,E1 -13295.72,E2 -13295.72} C_VEL
LIN {X 0,Y 354.66,Z 396.314,A -85,B 0,C 180,E1 -13296.651,E2 -13296.651} C_VEL
LIN {X 0,Y 354.812,Z 396.293,A -85,B 0,C 180,E1 -13299.112,E2 -13299.112} C_VEL
LIN {X 0,Y 354.894,Z 396.278,A -85,B 0,C 180,E1 -13302.72,E2 -13302.72} C_VEL
LIN {X 0,Y 354.947,Z 396.274,A -85,B 0,C 180,E1 -13306.255,E2 -13306.255} C_VEL
LIN {X 0,Y 354.974,Z 396.27,A -85,B 0,C 180,E1 -13309.736,E2 -13309.736} C_VEL
LIN {X 0,Y 355.121,Z 396.251,A -85,B 0,C 180,E1 -13313.18,E2 -13313.18} C_VEL
LIN {X 0,Y 355.241,Z 396.234,A -85,B 0,C 180,E1 -13317.732,E2 -13317.732} C_VEL
LIN {X 0,Y 355.392,Z 396.214,A -85,B 0,C 180,E1 -13320,E2 -13320} C_VEL
LIN {X 0,Y 355.241,Z 396.233,A -85,B 0,C 180,E1 -13322.268,E2 -13322.268} C_VEL
LIN {X 0,Y 355.121,Z 396.251,A -85,B 0,C 180,E1 -13326.819,E2 -13326.819} C_VEL
LIN {X 0,Y 354.973,Z 396.266,A -85,B 0,C 180,E1 -13330.264,E2 -13330.264} C_VEL
LIN {X 0,Y 354.938,Z 396.272,A -85,B 0,C 180,E1 -13334.019,E2 -13334.019} C_VEL
LIN {X 0,Y 354.919,Z 396.275,A -85,B 0,C 180,E1 -13338.109,E2 -13338.109} C_VEL
LIN {X 0,Y 354.83,Z 396.287,A -85,B 0,C 180,E1 -13342.106,E2 -13342.106} C_VEL
LIN {X 0,Y 354.895,Z 396.278,A -85,B 0,C 180,E1 -13345.828,E2 -13345.828} C_VEL
LIN {X 0,Y 354.814,Z 396.291,A -85,B 0,C 180,E1 -13349.682,E2 -13349.682} C_VEL
LIN {X 0,Y 354.803,Z 396.294,A -85,B 0,C 180,E1 -13353.702,E2 -13353.702} C_VEL
LIN {X 0,Y 354.796,Z 396.295,A -85,B 0,C 180,E1 -13356.46,E2 -13356.46} C_VEL
LIN {X 0,Y 354.822,Z 396.292,A -85,B 0,C 180,E1 -13359.424,E2 -13359.424} C_VEL
LIN {X 0,Y 354.835,Z 396.342,A -85,B 0,C 180,E1 -13362.331,E2 -13362.331} C_VEL
LIN {X 0,Y 355.764,Z 401.519,A -85,B 0,C 180,E1 -13366.259,E2 -13366.259} C_VEL
LIN {X 0,Y 356.601,Z 406.136,A -85,B 0,C 180,E1 -13369.431,E2 -13369.431} C_VEL
LIN {X 0,Y 357.378,Z 410.898,A -85,B 0,C 180,E1 -13372.438,E2 -13372.438} C_VEL
LIN {X 0,Y 357.343,Z 414.517,A -85,B 0,C 180,E1 -13374.537,E2 -13374.537} C_VEL
LIN {X 0,Y 356.507,Z 420.842,A -85,B 0,C 180,E1 -13377.96,E2 -13377.96} C_VEL
LIN {X 0,Y 355.814,Z 426.855,A -85,B 0,C 180,E1 -13381.058,E2 -13381.058} C_VEL
LIN {X 0,Y 355.066,Z 434.443,A -85,B 0,C 180,E1 -13384.814,E2 -13384.814} C_VEL
LIN {X 0,Y 354.478,Z 442.569,A -85,B 0,C 180,E1 -13388.724,E2 -13388.724} C_VEL
LIN {X 0,Y 354.393,Z 443.831,A -85,B 0,C 180,E1 -13389.318,E2 -13389.318} C_VEL
LIN {X 0,Y 357.073,Z 457.798,A -85,B 0,C 180,E1 -13389.997,E2 -13389.997} C_VEL
LIN {X 0,Y 358.63,Z 470.373,A -85,B 0,C 180,E1 -13390.79,E2 -13390.79} C_VEL
LIN {X 0,Y 359.842,Z 482.856,A -85,B 0,C 180,E1 -13391.791,E2 -13391.791} C_VEL
LIN {X 0,Y 358.803,Z 493.614,A -85,B 0,C 180,E1 -13392.767,E2 -13392.767} C_VEL
LIN {X 0,Y 357.588,Z 504.659,A -85,B 0,C 180,E1 -13394.029,E2 -13394.029} C_VEL
LIN {X 0,Y 356.572,Z 514.565,A -85,B 0,C 180,E1 -13395.445,E2 -13395.445} C_VEL
LIN {X 0,Y 355.454,Z 524.207,A -85,B 0,C 180,E1 -13397.148,E2 -13397.148} C_VEL
LIN {X 0,Y 354.554,Z 531.905,A -85,B 0,C 180,E1 -13398.857,E2 -13398.857} C_VEL
LIN {X 0,Y 354.08,Z 537.203,A -85,B 0,C 180,E1 -13400.287,E2 -13400.287} C_VEL
LIN {X 0,Y 353.653,Z 542.348,A -85,B 0,C 180,E1 -13402.004,E2 -13402.004} C_VEL
LIN {X 0,Y 353.435,Z 546.603,A -85,B 0,C 180,E1 -13403.851,E2 -13403.851} C_VEL
LIN {X 0,Y 353.357,Z 549.325,A -85,B 0,C 180,E1 -13405.437,E2 -13405.437} C_VEL
LIN {X 0,Y 353.318,Z 551.751,A -85,B 0,C 180,E1 -13407.72,E2 -13407.72} C_VEL
LIN {X 0,Y 353.4,Z 552.376,A -85,B 0,C 180,E1 -13408.86,E2 -13408.86} C_VEL
LIN {X 0,Y 353.411,Z 552.58,A -85,B 0,C 180,E1 -13410,E2 -13410} C_VEL
LIN {X 0,Y 353.42,Z 552.353,A -85,B 0,C 180,E1 -13411.139,E2 -13411.139} C_VEL
LIN {X 0,Y 353.333,Z 551.728,A -85,B 0,C 180,E1 -13412.28,E2 -13412.28} C_VEL
LIN {X 0,Y 353.283,Z 550.71,A -85,B 0,C 180,E1 -13413.421,E2 -13413.421} C_VEL
LIN {X 0,Y 353.36,Z 549.269,A -85,B 0,C 180,E1 -13414.563,E2 -13414.563} C_VEL
LIN {X 0,Y 353.446,Z 546.495,A -85,B 0,C 180,E1 -13416.166,E2 -13416.166} C_VEL
LIN {X 0,Y 353.653,Z 542.213,A -85,B 0,C 180,E1 -13417.996,E2 -13417.996} C_VEL
LIN {X 0,Y 354.202,Z 535.973,A -85,B 0,C 180,E1 -13419.998,E2 -13419.998} C_VEL
LIN {X 0,Y 354.8,Z 529.171,A -85,B 0,C 180,E1 -13421.714,E2 -13421.714} C_VEL
LIN {X 0,Y 355.81,Z 520.744,A -85,B 0,C 180,E1 -13423.419,E2 -13423.419} C_VEL
LIN {X 0,Y 356.771,Z 512.06,A -85,B 0,C 180,E1 -13424.837,E2 -13424.837} C_VEL
LIN {X 0,Y 357.749,Z 501.371,A -85,B 0,C 180,E1 -13426.256,E2 -13426.256} C_VEL
LIN {X 0,Y 358.904,Z 490.801,A -85,B 0,C 180,E1 -13427.374,E2 -13427.374} C_VEL
LIN {X 0,Y 359.584,Z 482.699,A -85,B 0,C 180,E1 -13428.075,E2 -13428.075} C_VEL
LIN {X 0,Y 358.296,Z 470.197,A -85,B 0,C 180,E1 -13429.045,E2 -13429.045} C_VEL
LIN {X 0,Y 356.498,Z 457.203,A -85,B 0,C 180,E1 -13429.824,E2 -13429.824} C_VEL
LIN {X 0,Y 354.383,Z 444.842,A -85,B 0,C 180,E1 -13430.382,E2 -13430.382} C_VEL
LIN {X 0,Y 354.886,Z 437.533,A -85,B 0,C 180,E1 -13433.865,E2 -13433.865} C_VEL
LIN {X 0,Y 355.47,Z 430.73,A -85,B 0,C 180,E1 -13437.165,E2 -13437.165} C_VEL
LIN {X 0,Y 356.138,Z 424.592,A -85,B 0,C 180,E1 -13440.224,E2 -13440.224} C_VEL
LIN {X 0,Y 356.864,Z 418.256,A -85,B 0,C 180,E1 -13443.464,E2 -13443.464} C_VEL
LIN {X 0,Y 357.446,Z 413.191,A -85,B 0,C 180,E1 -13446.145,E2 -13446.145} C_VEL
LIN {X 0,Y 357.258,Z 409.677,A -85,B 0,C 180,E1 -13448.105,E2 -13448.105} C_VEL
LIN {X 0,Y 356.239,Z 404.112,A -85,B 0,C 180,E1 -13451.437,E2 -13451.437} C_VEL
LIN {X 0,Y 355.138,Z 397.859,A -85,B 0,C 180,E1 -13455.431,E2 -13455.431} C_VEL
LIN {X 0,Y 354.824,Z 396.289,A -85,B 0,C 180,E1 -13456.531,E2 -13456.531} C_VEL
LIN {X 0,Y 354.82,Z 396.289,A -85,B 0,C 180,E1 -13459.183,E2 -13459.183} C_VEL
LIN {X 0,Y 354.804,Z 396.29,A -85,B 0,C 180,E1 -13462.401,E2 -13462.401} C_VEL
LIN {X 0,Y 354.807,Z 396.292,A -85,B 0,C 180,E1 -13464.94,E2 -13464.94} C_VEL
LIN {X 0,Y 354.786,Z 396.29,A -85,B 0,C 180,E1 -13468.405,E2 -13468.405} C_VEL
LIN {X 0,Y 354.84,Z 396.282,A -85,B 0,C 180,E1 -13471.618,E2 -13471.618} C_VEL
LIN {X 0,Y 354.892,Z 396.276,A -85,B 0,C 180,E1 -13474.172,E2 -13474.172} C_VEL
LIN {X 0,Y 354.827,Z 396.283,A -85,B 0,C 180,E1 -13477.894,E2 -13477.894} C_VEL
LIN {X 0,Y 354.915,Z 396.272,A -85,B 0,C 180,E1 -13481.891,E2 -13481.891} C_VEL
LIN {X 0,Y 354.935,Z 396.27,A -85,B 0,C 180,E1 -13485.981,E2 -13485.981} C_VEL
LIN {X 0,Y 354.97,Z 396.265,A -85,B 0,C 180,E1 -13489.736,E2 -13489.736} C_VEL
LIN {X 0,Y 355.118,Z 396.249,A -85,B 0,C 180,E1 -13493.18,E2 -13493.18} C_VEL
LIN {X 0,Y 355.238,Z 396.232,A -85,B 0,C 180,E1 -13497.732,E2 -13497.732} C_VEL
LIN {X 0,Y 355.391,Z 396.214,A -85,B 0,C 180,E1 -13500,E2 -13500} C_VEL
LIN {X 0,Y 355.238,Z 396.235,A -85,B 0,C 180,E1 -13502.268,E2 -13502.268} C_VEL
LIN {X 0,Y 355.13,Z 396.249,A -85,B 0,C 180,E1 -13506.82,E2 -13506.82} C_VEL
LIN {X 0,Y 355.007,Z 396.262,A -85,B 0,C 180,E1 -13509.113,E2 -13509.113} C_VEL
LIN {X 0,Y 354.914,Z 396.278,A -85,B 0,C 180,E1 -13512.581,E2 -13512.581} C_VEL
LIN {X 0,Y 354.882,Z 396.279,A -85,B 0,C 180,E1 -13516.097,E2 -13516.097} C_VEL
LIN {X 0,Y 354.899,Z 396.28,A -85,B 0,C 180,E1 -13518.472,E2 -13518.472} C_VEL
LIN {X 0,Y 354.828,Z 396.287,A -85,B 0,C 180,E1 -13522.107,E2 -13522.107} C_VEL
LIN {X 0,Y 354.893,Z 396.276,A -85,B 0,C 180,E1 -13525.828,E2 -13525.828} C_VEL
LIN {X 0,Y 354.848,Z 396.282,A -85,B 0,C 180,E1 -13529.679,E2 -13529.679} C_VEL
LIN {X 0,Y 354.801,Z 396.288,A -85,B 0,C 180,E1 -13533.703,E2 -13533.703} C_VEL
LIN {X 0,Y 354.795,Z 396.291,A -85,B 0,C 180,E1 -13536.46,E2 -13536.46} C_VEL
